ABB RAPID module: P401.mod

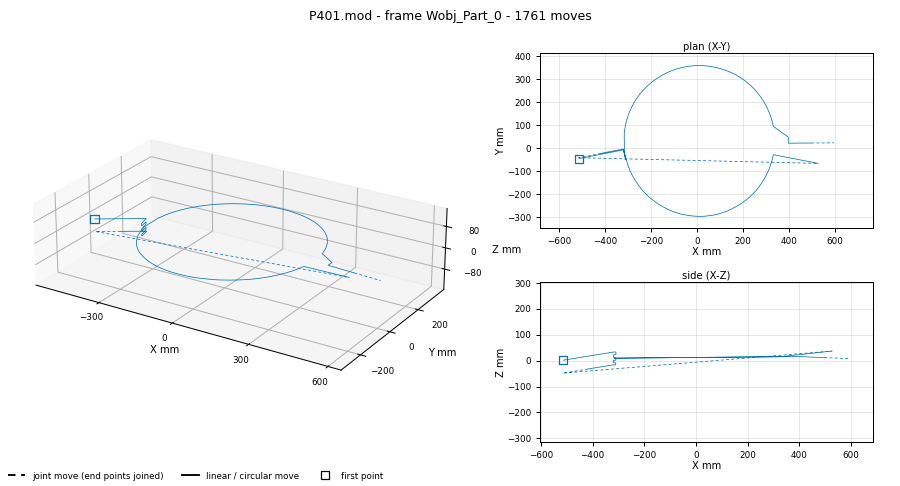
[picture p0: tool path of P401.mod in frame Wobj_Part_0, 1761 of 1771 moves have a stored position in this frame; points joined in program order, loops and branches not executed]
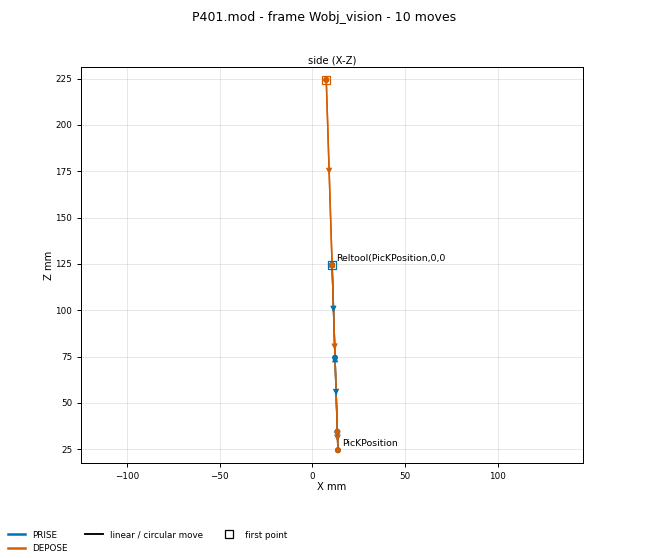
[picture p1: tool path of P401.mod in frame Wobj_vision, 10 of 1771 moves have a stored position in this frame; points joined in program order, loops and branches not executed]
MODULE P401

    ! Nom         :P401
    ! Description :
    ! Créé le     :07/06/2023 14:41:53

    LOCAL CONST SPEEDDATA VitesseLente :=[10,500,0,0];
	LOCAL CONST SPEEDDATA VitesseRapide :=[30,500,0,0];
	LOCAL CONST SPEEDDATA VitesseTronconnage :=[2,500,0,0];
	LOCAL CONST SPEEDDATA VitesseTronconnageApp :=[10,500,0,0];
    !
    !Point de prise
    LOCAL PERS Robtarget PicKPosition := [[13.7351915229446,28.8988205963881,24.4259709392431],[0.015425718644535,0.66713477772881,0.744749815337416,0.00639907055097392],[0,0,0,0],[8.999999E+09,8.999999E+09,8.999999E+09,8.999999E+09,8.999999E+09,8.999999E+09]];
	LOCAL PERS Pose Ref := [[0,0,0],[1,0,0,0]];
    !
    !Declaration des points de meulage

    !Tr_meulage_motif_1 : Meulage d'un motif
    LOCAL CONST Robtarget Tr_meulage_motif_1_0 := [[-319.4905625,-7.31827685546875,33.72298046875],[0.588012732058927,-0.500859688362471,0.411836559206125,-0.483498963816164],[0,0,0,0],[8.999999E+09,8.999999E+09,8.999999E+09,8.999999E+09,8.999999E+09,8.999999E+09]];
    LOCAL CONST Robtarget Tr_meulage_motif_1_1 := [[-319.26584375,-8.29269921875,33.72351171875],[0.588012732058927,-0.500859688362471,0.411836559206125,-0.483498963816164],[0,0,0,0],[8.999999E+09,8.999999E+09,8.999999E+09,8.999999E+09,8.999999E+09,8.999999E+09]];
    LOCAL CONST Robtarget Tr_meulage_motif_1_2 := [[-319.041125,-9.26712109375,33.72404296875],[0.588012732058927,-0.500859688362471,0.411836559206125,-0.483498963816164],[0,0,0,0],[8.999999E+09,8.999999E+09,8.999999E+09,8.999999E+09,8.999999E+09,8.999999E+09]];
    LOCAL CONST Robtarget Tr_meulage_motif_1_3 := [[-318.81640625,-10.24154296875,33.72457421875],[0.588012732058927,-0.500859688362471,0.411836559206125,-0.483498963816164],[0,0,0,0],[8.999999E+09,8.999999E+09,8.999999E+09,8.999999E+09,8.999999E+09,8.999999E+09]];
    LOCAL CONST Robtarget Tr_meulage_motif_1_4 := [[-318.59165625,-11.21596484375,33.725109375],[0.588012732058927,-0.500859688362471,0.411836559206125,-0.483498963816164],[0,0,0,0],[8.999999E+09,8.999999E+09,8.999999E+09,8.999999E+09,8.999999E+09,8.999999E+09]];
    LOCAL CONST Robtarget Tr_meulage_motif_1_5 := [[-318.3669375,-12.1903876953125,33.725640625],[0.588012732058927,-0.500859688362471,0.411836559206125,-0.483498963816164],[0,0,0,0],[8.999999E+09,8.999999E+09,8.999999E+09,8.999999E+09,8.999999E+09,8.999999E+09]];
    LOCAL CONST Robtarget Tr_meulage_motif_1_6 := [[-318.14221875,-13.1648095703125,33.726171875],[0.588012732058927,-0.500859688362471,0.411836559206125,-0.483498963816164],[0,0,0,0],[8.999999E+09,8.999999E+09,8.999999E+09,8.999999E+09,8.999999E+09,8.999999E+09]];
    LOCAL CONST Robtarget Tr_meulage_motif_1_7 := [[-317.9175,-14.1392314453125,33.726703125],[0.588012732058927,-0.500859688362471,0.411836559206125,-0.483498963816164],[0,0,0,0],[8.999999E+09,8.999999E+09,8.999999E+09,8.999999E+09,8.999999E+09,8.999999E+09]];
    LOCAL CONST Robtarget Tr_meulage_motif_1_8 := [[-317.69278125,-15.1136533203125,33.727234375],[0.588012732058927,-0.500859688362471,0.411836559206125,-0.483498963816164],[0,0,0,0],[8.999999E+09,8.999999E+09,8.999999E+09,8.999999E+09,8.999999E+09,8.999999E+09]];
    LOCAL CONST Robtarget Tr_meulage_motif_1_9 := [[-317.46803125,-16.0880751953125,33.72776953125],[0.588012732058927,-0.500859688362471,0.411836559206125,-0.483498963816164],[0,0,0,0],[8.999999E+09,8.999999E+09,8.999999E+09,8.999999E+09,8.999999E+09,8.999999E+09]];
    LOCAL CONST Robtarget Tr_meulage_motif_1_10 := [[-317.2433125,-17.062498046875,33.72830078125],[0.588012732058927,-0.500859688362471,0.411836559206125,-0.483498963816164],[0,0,0,0],[8.999999E+09,8.999999E+09,8.999999E+09,8.999999E+09,8.999999E+09,8.999999E+09]];
    LOCAL CONST Robtarget Tr_meulage_motif_1_11 := [[-317.01859375,-18.036919921875,33.72883203125],[0.588012732058927,-0.500859688362471,0.411836559206125,-0.483498963816164],[0,0,0,0],[8.999999E+09,8.999999E+09,8.999999E+09,8.999999E+09,8.999999E+09,8.999999E+09]];
    LOCAL CONST Robtarget Tr_meulage_motif_1_12 := [[-316.793875,-19.011341796875,33.72936328125],[0.588012732058927,-0.500859688362471,0.411836559206125,-0.483498963816164],[0,0,0,0],[8.999999E+09,8.999999E+09,8.999999E+09,8.999999E+09,8.999999E+09,8.999999E+09]];
    LOCAL CONST Robtarget Tr_meulage_motif_1_13 := [[-316.56915625,-19.985763671875,33.7298984375],[0.588012732058927,-0.500859688362471,0.411836559206125,-0.483498963816164],[0,0,0,0],[8.999999E+09,8.999999E+09,8.999999E+09,8.999999E+09,8.999999E+09,8.999999E+09]];
    LOCAL CONST Robtarget Tr_meulage_motif_1_14 := [[-316.34440625,-20.960185546875,33.7304296875],[0.588012732058927,-0.500859688362471,0.411836559206125,-0.483498963816164],[0,0,0,0],[8.999999E+09,8.999999E+09,8.999999E+09,8.999999E+09,8.999999E+09,8.999999E+09]];
    LOCAL CONST Robtarget Tr_meulage_motif_1_15 := [[-316.1196875,-21.934607421875,33.7309609375],[0.588012732058927,-0.500859688362471,0.411836559206125,-0.483498963816164],[0,0,0,0],[8.999999E+09,8.999999E+09,8.999999E+09,8.999999E+09,8.999999E+09,8.999999E+09]];
    LOCAL CONST Robtarget Tr_meulage_motif_1_16 := [[-315.89496875,-22.909029296875,33.7314921875],[0.588012732058927,-0.500859688362471,0.411836559206125,-0.483498963816164],[0,0,0,0],[8.999999E+09,8.999999E+09,8.999999E+09,8.999999E+09,8.999999E+09,8.999999E+09]];
    LOCAL CONST Robtarget Tr_meulage_motif_1_17 := [[-315.67025,-23.883451171875,33.73202734375],[0.588012732058927,-0.500859688362471,0.411836559206125,-0.483498963816164],[0,0,0,0],[8.999999E+09,8.999999E+09,8.999999E+09,8.999999E+09,8.999999E+09,8.999999E+09]];
    LOCAL CONST Robtarget Tr_meulage_motif_1_18 := [[-315.44553125,-24.857875,33.73255859375],[0.588012732058927,-0.500859688362471,0.411836559206125,-0.483498963816164],[0,0,0,0],[8.999999E+09,8.999999E+09,8.999999E+09,8.999999E+09,8.999999E+09,8.999999E+09]];
    LOCAL CONST Robtarget Tr_meulage_motif_1_19 := [[-315.22078125,-25.832296875,33.73308984375],[0.588012732058927,-0.500859688362471,0.411836559206125,-0.483498963816164],[0,0,0,0],[8.999999E+09,8.999999E+09,8.999999E+09,8.999999E+09,8.999999E+09,8.999999E+09]];
    LOCAL CONST Robtarget Tr_meulage_motif_1_20 := [[-314.9960625,-26.80671875,33.73362109375],[0.588012732058927,-0.500859688362471,0.411836559206125,-0.483498963816164],[0,0,0,0],[8.999999E+09,8.999999E+09,8.999999E+09,8.999999E+09,8.999999E+09,8.999999E+09]];
    LOCAL CONST Robtarget Tr_meulage_motif_1_21 := [[-314.77134375,-27.781140625,33.73415234375],[0.588012732058927,-0.500859688362471,0.411836559206125,-0.483498963816164],[0,0,0,0],[8.999999E+09,8.999999E+09,8.999999E+09,8.999999E+09,8.999999E+09,8.999999E+09]];
    LOCAL CONST Robtarget Tr_meulage_motif_1_22 := [[-314.546625,-28.7555625,33.7346875],[0.588012732058927,-0.500859688362471,0.411836559206125,-0.483498963816164],[0,0,0,0],[8.999999E+09,8.999999E+09,8.999999E+09,8.999999E+09,8.999999E+09,8.999999E+09]];
    LOCAL CONST Robtarget Tr_meulage_motif_1_23 := [[-314.32190625,-29.729984375,33.73521875],[0.588012732058927,-0.500859688362471,0.411836559206125,-0.483498963816164],[0,0,0,0],[8.999999E+09,8.999999E+09,8.999999E+09,8.999999E+09,8.999999E+09,8.999999E+09]];
    LOCAL CONST Robtarget Tr_meulage_motif_1_24 := [[-314.09715625,-30.70440625,33.73575],[0.588012732058927,-0.500859688362471,0.411836559206125,-0.483498963816164],[0,0,0,0],[8.999999E+09,8.999999E+09,8.999999E+09,8.999999E+09,8.999999E+09,8.999999E+09]];
    LOCAL CONST Robtarget Tr_meulage_motif_1_25 := [[-313.8724375,-31.678828125,33.73628125],[0.588012732058927,-0.500859688362471,0.411836559206125,-0.483498963816164],[0,0,0,0],[8.999999E+09,8.999999E+09,8.999999E+09,8.999999E+09,8.999999E+09,8.999999E+09]];
    LOCAL CONST Robtarget Tr_meulage_motif_1_26 := [[-313.64771875,-32.65325,33.73681640625],[0.588012732058927,-0.500859688362471,0.411836559206125,-0.483498963816164],[0,0,0,0],[8.999999E+09,8.999999E+09,8.999999E+09,8.999999E+09,8.999999E+09,8.999999E+09]];
    LOCAL CONST Robtarget Tr_meulage_motif_1_27 := [[-313.423,-33.627671875,33.73734765625],[0.588012732058927,-0.500859688362471,0.411836559206125,-0.483498963816164],[0,0,0,0],[8.999999E+09,8.999999E+09,8.999999E+09,8.999999E+09,8.999999E+09,8.999999E+09]];
    LOCAL CONST Robtarget Tr_meulage_motif_1_28 := [[-313.19828125,-34.60209375,33.73787890625],[0.588012732058927,-0.500859688362471,0.411836559206125,-0.483498963816164],[0,0,0,0],[8.999999E+09,8.999999E+09,8.999999E+09,8.999999E+09,8.999999E+09,8.999999E+09]];
    LOCAL CONST Robtarget Tr_meulage_motif_1_29 := [[-312.97353125,-35.576515625,33.73841015625],[0.588012732058927,-0.500859688362471,0.411836559206125,-0.483498963816164],[0,0,0,0],[8.999999E+09,8.999999E+09,8.999999E+09,8.999999E+09,8.999999E+09,8.999999E+09]];
    LOCAL CONST Robtarget Tr_meulage_motif_1_30 := [[-312.7488125,-36.5509375,33.73894140625],[0.588012732058927,-0.500859688362471,0.411836559206125,-0.483498963816164],[0,0,0,0],[8.999999E+09,8.999999E+09,8.999999E+09,8.999999E+09,8.999999E+09,8.999999E+09]];
    LOCAL CONST Robtarget Tr_meulage_motif_1_31 := [[-312.52409375,-37.525359375,33.7394765625],[0.588012732058927,-0.500859688362471,0.411836559206125,-0.483498963816164],[0,0,0,0],[8.999999E+09,8.999999E+09,8.999999E+09,8.999999E+09,8.999999E+09,8.999999E+09]];
    LOCAL CONST Robtarget Tr_meulage_motif_1_32 := [[-312.299375,-38.49978125,33.7400078125],[0.588012732058927,-0.500859688362471,0.411836559206125,-0.483498963816164],[0,0,0,0],[8.999999E+09,8.999999E+09,8.999999E+09,8.999999E+09,8.999999E+09,8.999999E+09]];
    LOCAL CONST Robtarget Tr_meulage_motif_1_33 := [[-312.07465625,-39.47420703125,33.7405390625],[0.588012732058927,-0.500859688362471,0.411836559206125,-0.483498963816164],[0,0,0,0],[8.999999E+09,8.999999E+09,8.999999E+09,8.999999E+09,8.999999E+09,8.999999E+09]];
    LOCAL CONST Robtarget Tr_meulage_motif_1_34 := [[-311.84990625,-40.44862890625,33.7410703125],[0.588012732058927,-0.500859688362471,0.411836559206125,-0.483498963816164],[0,0,0,0],[8.999999E+09,8.999999E+09,8.999999E+09,8.999999E+09,8.999999E+09,8.999999E+09]];
    LOCAL CONST Robtarget Tr_meulage_motif_1_35 := [[-311.6251875,-41.42305078125,33.74160546875],[0.588012732058927,-0.500859688362471,0.411836559206125,-0.483498963816164],[0,0,0,0],[8.999999E+09,8.999999E+09,8.999999E+09,8.999999E+09,8.999999E+09,8.999999E+09]];
    LOCAL CONST Robtarget Tr_meulage_motif_1_36 := [[-311.40046875,-42.39747265625,33.74213671875],[0.588012732058927,-0.500859688362471,0.411836559206125,-0.483498963816164],[0,0,0,0],[8.999999E+09,8.999999E+09,8.999999E+09,8.999999E+09,8.999999E+09,8.999999E+09]];
    LOCAL CONST Robtarget Tr_meulage_motif_1_37 := [[-311.17575,-43.37189453125,33.74266796875],[0.588012732058927,-0.500859688362471,0.411836559206125,-0.483498963816164],[0,0,0,0],[8.999999E+09,8.999999E+09,8.999999E+09,8.999999E+09,8.999999E+09,8.999999E+09]];
    LOCAL CONST Robtarget Tr_meulage_motif_1_38 := [[-310.95103125,-44.34631640625,33.74319921875],[0.588012732058927,-0.500859688362471,0.411836559206125,-0.483498963816164],[0,0,0,0],[8.999999E+09,8.999999E+09,8.999999E+09,8.999999E+09,8.999999E+09,8.999999E+09]];
    LOCAL CONST Robtarget Tr_meulage_motif_1_39 := [[-310.72928125,-45.31385546875,33.63314453125],[0.588012732058927,-0.500859688362471,0.411836559206125,-0.483498963816164],[0,0,0,0],[8.999999E+09,8.999999E+09,8.999999E+09,8.999999E+09,8.999999E+09,8.999999E+09]];
    LOCAL CONST Robtarget Tr_meulage_motif_1_40 := [[-310.51909375,-46.23683984375,33.4224765625],[0.588012732058927,-0.500859688362471,0.411836559206125,-0.483498963816164],[0,0,0,0],[8.999999E+09,8.999999E+09,8.999999E+09,8.999999E+09,8.999999E+09,8.999999E+09]];
    LOCAL CONST Robtarget Tr_meulage_motif_1_41 := [[-310.3306875,-47.06864453125,33.15110546875],[0.588012732058927,-0.500859688362471,0.411836559206125,-0.483498963816164],[0,0,0,0],[8.999999E+09,8.999999E+09,8.999999E+09,8.999999E+09,8.999999E+09,8.999999E+09]];
    LOCAL CONST Robtarget Tr_meulage_motif_1_42 := [[-310.16546875,-47.8003046875,32.87558984375],[0.588012732058927,-0.500859688362471,0.411836559206125,-0.483498963816164],[0,0,0,0],[8.999999E+09,8.999999E+09,8.999999E+09,8.999999E+09,8.999999E+09,8.999999E+09]];
    LOCAL CONST Robtarget Tr_meulage_motif_1_43 := [[-309.92534375,-48.875234375,32.26009765625],[0.588012732058927,-0.500859688362471,0.411836559206125,-0.483498963816164],[0,0,0,0],[8.999999E+09,8.999999E+09,8.999999E+09,8.999999E+09,8.999999E+09,8.999999E+09]];
    LOCAL CONST Robtarget Tr_meulage_motif_1_44 := [[-309.70534375,-49.8757109375,31.41305078125],[0.588012732058927,-0.500859688362471,0.411836559206125,-0.483498963816164],[0,0,0,0],[8.999999E+09,8.999999E+09,8.999999E+09,8.999999E+09,8.999999E+09,8.999999E+09]];
    LOCAL CONST Robtarget Tr_meulage_motif_1_45 := [[-309.5270625,-50.7050546875,30.389705078125],[0.588012732058927,-0.500859688362471,0.411836559206125,-0.483498963816164],[0,0,0,0],[8.999999E+09,8.999999E+09,8.999999E+09,8.999999E+09,8.999999E+09,8.999999E+09]];
    LOCAL CONST Robtarget Tr_meulage_motif_1_46 := [[-309.430625,-51.1843984375,29.273861328125],[0.588012732058927,-0.500859688362471,0.411836559206125,-0.483498963816164],[0,0,0,0],[8.999999E+09,8.999999E+09,8.999999E+09,8.999999E+09,8.999999E+09,8.999999E+09]];
    LOCAL CONST Robtarget Tr_meulage_motif_1_47 := [[-309.43284375,-51.2130625,28.5779609375],[0.588012732058927,-0.500859688362471,0.411836559206125,-0.483498963816164],[0,0,0,0],[8.999999E+09,8.999999E+09,8.999999E+09,8.999999E+09,8.999999E+09,8.999999E+09]];
    LOCAL CONST Robtarget Tr_meulage_motif_1_48 := [[-309.44071875,-51.21523828125,27.91676171875],[0.588012732058927,-0.500859688362471,0.411836559206125,-0.483498963816164],[0,0,0,0],[8.999999E+09,8.999999E+09,8.999999E+09,8.999999E+09,8.999999E+09,8.999999E+09]];
    LOCAL CONST Robtarget Tr_meulage_motif_1_49 := [[-309.46090625,-51.16394140625,27.2556875],[0.588012732058927,-0.500859688362471,0.411836559206125,-0.483498963816164],[0,0,0,0],[8.999999E+09,8.999999E+09,8.999999E+09,8.999999E+09,8.999999E+09,8.999999E+09]];
    LOCAL CONST Robtarget Tr_meulage_motif_1_50 := [[-309.586,-50.68209375,26.1537578125],[0.588012732058927,-0.500859688362471,0.411836559206125,-0.483498963816164],[0,0,0,0],[8.999999E+09,8.999999E+09,8.999999E+09,8.999999E+09,8.999999E+09,8.999999E+09]];
    LOCAL CONST Robtarget Tr_meulage_motif_1_51 := [[-309.79046875,-49.85069140625,25.14675390625],[0.588012732058927,-0.500859688362471,0.411836559206125,-0.483498963816164],[0,0,0,0],[8.999999E+09,8.999999E+09,8.999999E+09,8.999999E+09,8.999999E+09,8.999999E+09]];
    LOCAL CONST Robtarget Tr_meulage_motif_1_52 := [[-310.03034375,-48.85619140625,24.317396484375],[0.588012732058927,-0.500859688362471,0.411836559206125,-0.483498963816164],[0,0,0,0],[8.999999E+09,8.999999E+09,8.999999E+09,8.999999E+09,8.999999E+09,8.999999E+09]];
    LOCAL CONST Robtarget Tr_meulage_motif_1_53 := [[-310.1894375,-48.18797265625,23.921310546875],[0.588012732058927,-0.500859688362471,0.411836559206125,-0.483498963816164],[0,0,0,0],[8.999999E+09,8.999999E+09,8.999999E+09,8.999999E+09,8.999999E+09,8.999999E+09]];
    LOCAL CONST Robtarget Tr_meulage_motif_1_54 := [[-310.45553125,-47.061046875,23.433201171875],[0.588012732058927,-0.500859688362471,0.411836559206125,-0.483498963816164],[0,0,0,0],[8.999999E+09,8.999999E+09,8.999999E+09,8.999999E+09,8.999999E+09,8.999999E+09]];
    LOCAL CONST Robtarget Tr_meulage_motif_1_55 := [[-310.6485625,-46.23849609375,23.168677734375],[0.588012732058927,-0.500859688362471,0.411836559206125,-0.483498963816164],[0,0,0,0],[8.999999E+09,8.999999E+09,8.999999E+09,8.999999E+09,8.999999E+09,8.999999E+09]];
    LOCAL CONST Robtarget Tr_meulage_motif_1_56 := [[-310.8604375,-45.3310078125,22.963728515625],[0.588012732058927,-0.500859688362471,0.411836559206125,-0.483498963816164],[0,0,0,0],[8.999999E+09,8.999999E+09,8.999999E+09,8.999999E+09,8.999999E+09,8.999999E+09]];
    LOCAL CONST Robtarget Tr_meulage_motif_1_57 := [[-311.0823125,-44.37491015625,22.85462109375],[0.588012732058927,-0.500859688362471,0.411836559206125,-0.483498963816164],[0,0,0,0],[8.999999E+09,8.999999E+09,8.999999E+09,8.999999E+09,8.999999E+09,8.999999E+09]];
    LOCAL CONST Robtarget Tr_meulage_motif_1_58 := [[-311.3066875,-43.4081015625,22.7435078125],[0.588012732058927,-0.500859688362471,0.411836559206125,-0.483498963816164],[0,0,0,0],[8.999999E+09,8.999999E+09,8.999999E+09,8.999999E+09,8.999999E+09,8.999999E+09]];
    LOCAL CONST Robtarget Tr_meulage_motif_1_59 := [[-311.53140625,-42.4336796875,22.742974609375],[0.588012732058927,-0.500859688362471,0.411836559206125,-0.483498963816164],[0,0,0,0],[8.999999E+09,8.999999E+09,8.999999E+09,8.999999E+09,8.999999E+09,8.999999E+09]];
    LOCAL CONST Robtarget Tr_meulage_motif_1_60 := [[-311.756125,-41.4592578125,22.742443359375],[0.588012732058927,-0.500859688362471,0.411836559206125,-0.483498963816164],[0,0,0,0],[8.999999E+09,8.999999E+09,8.999999E+09,8.999999E+09,8.999999E+09,8.999999E+09]];
    LOCAL CONST Robtarget Tr_meulage_motif_1_61 := [[-311.980875,-40.48483203125,22.74191015625],[0.588012732058927,-0.500859688362471,0.411836559206125,-0.483498963816164],[0,0,0,0],[8.999999E+09,8.999999E+09,8.999999E+09,8.999999E+09,8.999999E+09,8.999999E+09]];
    LOCAL CONST Robtarget Tr_meulage_motif_1_62 := [[-312.20559375,-39.51041015625,22.74137890625],[0.588012732058927,-0.500859688362471,0.411836559206125,-0.483498963816164],[0,0,0,0],[8.999999E+09,8.999999E+09,8.999999E+09,8.999999E+09,8.999999E+09,8.999999E+09]];
    LOCAL CONST Robtarget Tr_meulage_motif_1_63 := [[-312.4303125,-38.53598828125,22.740845703125],[0.588012732058927,-0.500859688362471,0.411836559206125,-0.483498963816164],[0,0,0,0],[8.999999E+09,8.999999E+09,8.999999E+09,8.999999E+09,8.999999E+09,8.999999E+09]];
    LOCAL CONST Robtarget Tr_meulage_motif_1_64 := [[-312.65503125,-37.56156640625,22.740314453125],[0.588012732058927,-0.500859688362471,0.411836559206125,-0.483498963816164],[0,0,0,0],[8.999999E+09,8.999999E+09,8.999999E+09,8.999999E+09,8.999999E+09,8.999999E+09]];
    LOCAL CONST Robtarget Tr_meulage_motif_1_65 := [[-312.87975,-36.58714453125,22.739783203125],[0.588012732058927,-0.500859688362471,0.411836559206125,-0.483498963816164],[0,0,0,0],[8.999999E+09,8.999999E+09,8.999999E+09,8.999999E+09,8.999999E+09,8.999999E+09]];
    LOCAL CONST Robtarget Tr_meulage_motif_1_66 := [[-313.1045,-35.61272265625,22.73925],[0.588012732058927,-0.500859688362471,0.411836559206125,-0.483498963816164],[0,0,0,0],[8.999999E+09,8.999999E+09,8.999999E+09,8.999999E+09,8.999999E+09,8.999999E+09]];
    LOCAL CONST Robtarget Tr_meulage_motif_1_67 := [[-313.32921875,-34.63830078125,22.73871875],[0.588012732058927,-0.500859688362471,0.411836559206125,-0.483498963816164],[0,0,0,0],[8.999999E+09,8.999999E+09,8.999999E+09,8.999999E+09,8.999999E+09,8.999999E+09]];
    LOCAL CONST Robtarget Tr_meulage_motif_1_68 := [[-313.5539375,-33.66387890625,22.738185546875],[0.588012732058927,-0.500859688362471,0.411836559206125,-0.483498963816164],[0,0,0,0],[8.999999E+09,8.999999E+09,8.999999E+09,8.999999E+09,8.999999E+09,8.999999E+09]];
    LOCAL CONST Robtarget Tr_meulage_motif_1_69 := [[-313.77865625,-32.68945703125,22.737654296875],[0.588012732058927,-0.500859688362471,0.411836559206125,-0.483498963816164],[0,0,0,0],[8.999999E+09,8.999999E+09,8.999999E+09,8.999999E+09,8.999999E+09,8.999999E+09]];
    LOCAL CONST Robtarget Tr_meulage_motif_1_70 := [[-314.003375,-31.71503515625,22.73712109375],[0.588012732058927,-0.500859688362471,0.411836559206125,-0.483498963816164],[0,0,0,0],[8.999999E+09,8.999999E+09,8.999999E+09,8.999999E+09,8.999999E+09,8.999999E+09]];
    LOCAL CONST Robtarget Tr_meulage_motif_1_71 := [[-314.228125,-30.74061328125,22.73658984375],[0.588012732058927,-0.500859688362471,0.411836559206125,-0.483498963816164],[0,0,0,0],[8.999999E+09,8.999999E+09,8.999999E+09,8.999999E+09,8.999999E+09,8.999999E+09]];
    LOCAL CONST Robtarget Tr_meulage_motif_1_72 := [[-314.45284375,-29.76619140625,22.736056640625],[0.588012732058927,-0.500859688362471,0.411836559206125,-0.483498963816164],[0,0,0,0],[8.999999E+09,8.999999E+09,8.999999E+09,8.999999E+09,8.999999E+09,8.999999E+09]];
    LOCAL CONST Robtarget Tr_meulage_motif_1_73 := [[-314.6775625,-28.79176953125,22.735525390625],[0.588012732058927,-0.500859688362471,0.411836559206125,-0.483498963816164],[0,0,0,0],[8.999999E+09,8.999999E+09,8.999999E+09,8.999999E+09,8.999999E+09,8.999999E+09]];
    LOCAL CONST Robtarget Tr_meulage_motif_1_74 := [[-314.90228125,-27.81734765625,22.7349921875],[0.588012732058927,-0.500859688362471,0.411836559206125,-0.483498963816164],[0,0,0,0],[8.999999E+09,8.999999E+09,8.999999E+09,8.999999E+09,8.999999E+09,8.999999E+09]];
    LOCAL CONST Robtarget Tr_meulage_motif_1_75 := [[-315.12703125,-26.84292578125,22.7344609375],[0.588012732058927,-0.500859688362471,0.411836559206125,-0.483498963816164],[0,0,0,0],[8.999999E+09,8.999999E+09,8.999999E+09,8.999999E+09,8.999999E+09,8.999999E+09]];
    LOCAL CONST Robtarget Tr_meulage_motif_1_76 := [[-315.35175,-25.868501953125,22.7339296875],[0.588012732058927,-0.500859688362471,0.411836559206125,-0.483498963816164],[0,0,0,0],[8.999999E+09,8.999999E+09,8.999999E+09,8.999999E+09,8.999999E+09,8.999999E+09]];
    LOCAL CONST Robtarget Tr_meulage_motif_1_77 := [[-315.57646875,-24.894080078125,22.733396484375],[0.588012732058927,-0.500859688362471,0.411836559206125,-0.483498963816164],[0,0,0,0],[8.999999E+09,8.999999E+09,8.999999E+09,8.999999E+09,8.999999E+09,8.999999E+09]];
    LOCAL CONST Robtarget Tr_meulage_motif_1_78 := [[-315.8011875,-23.919658203125,22.732865234375],[0.588012732058927,-0.500859688362471,0.411836559206125,-0.483498963816164],[0,0,0,0],[8.999999E+09,8.999999E+09,8.999999E+09,8.999999E+09,8.999999E+09,8.999999E+09]];
    LOCAL CONST Robtarget Tr_meulage_motif_1_79 := [[-316.02590625,-22.945236328125,22.73233203125],[0.588012732058927,-0.500859688362471,0.411836559206125,-0.483498963816164],[0,0,0,0],[8.999999E+09,8.999999E+09,8.999999E+09,8.999999E+09,8.999999E+09,8.999999E+09]];
    LOCAL CONST Robtarget Tr_meulage_motif_1_80 := [[-316.25065625,-21.970814453125,22.73180078125],[0.588012732058927,-0.500859688362471,0.411836559206125,-0.483498963816164],[0,0,0,0],[8.999999E+09,8.999999E+09,8.999999E+09,8.999999E+09,8.999999E+09,8.999999E+09]];
    LOCAL CONST Robtarget Tr_meulage_motif_1_81 := [[-316.475375,-20.996392578125,22.731267578125],[0.588012732058927,-0.500859688362471,0.411836559206125,-0.483498963816164],[0,0,0,0],[8.999999E+09,8.999999E+09,8.999999E+09,8.999999E+09,8.999999E+09,8.999999E+09]];
    LOCAL CONST Robtarget Tr_meulage_motif_1_82 := [[-316.70009375,-20.021970703125,22.730736328125],[0.588012732058927,-0.500859688362471,0.411836559206125,-0.483498963816164],[0,0,0,0],[8.999999E+09,8.999999E+09,8.999999E+09,8.999999E+09,8.999999E+09,8.999999E+09]];
    LOCAL CONST Robtarget Tr_meulage_motif_1_83 := [[-316.9248125,-19.047548828125,22.730203125],[0.588012732058927,-0.500859688362471,0.411836559206125,-0.483498963816164],[0,0,0,0],[8.999999E+09,8.999999E+09,8.999999E+09,8.999999E+09,8.999999E+09,8.999999E+09]];
    LOCAL CONST Robtarget Tr_meulage_motif_1_84 := [[-317.14953125,-18.073126953125,22.729671875],[0.588012732058927,-0.500859688362471,0.411836559206125,-0.483498963816164],[0,0,0,0],[8.999999E+09,8.999999E+09,8.999999E+09,8.999999E+09,8.999999E+09,8.999999E+09]];
    LOCAL CONST Robtarget Tr_meulage_motif_1_85 := [[-317.37428125,-17.098705078125,22.729138671875],[0.588012732058927,-0.500859688362471,0.411836559206125,-0.483498963816164],[0,0,0,0],[8.999999E+09,8.999999E+09,8.999999E+09,8.999999E+09,8.999999E+09,8.999999E+09]];
    LOCAL CONST Robtarget Tr_meulage_motif_1_86 := [[-317.599,-16.1242822265625,22.728607421875],[0.588012732058927,-0.500859688362471,0.411836559206125,-0.483498963816164],[0,0,0,0],[8.999999E+09,8.999999E+09,8.999999E+09,8.999999E+09,8.999999E+09,8.999999E+09]];
    LOCAL CONST Robtarget Tr_meulage_motif_1_87 := [[-317.82371875,-15.1498603515625,22.72807421875],[0.588012732058927,-0.500859688362471,0.411836559206125,-0.483498963816164],[0,0,0,0],[8.999999E+09,8.999999E+09,8.999999E+09,8.999999E+09,8.999999E+09,8.999999E+09]];
    LOCAL CONST Robtarget Tr_meulage_motif_1_88 := [[-318.0484375,-14.1754384765625,22.72754296875],[0.588012732058927,-0.500859688362471,0.411836559206125,-0.483498963816164],[0,0,0,0],[8.999999E+09,8.999999E+09,8.999999E+09,8.999999E+09,8.999999E+09,8.999999E+09]];
    LOCAL CONST Robtarget Tr_meulage_motif_1_89 := [[-318.2728125,-13.208626953125,22.6164296875],[0.588012732058927,-0.500859688362471,0.411836559206125,-0.483498963816164],[0,0,0,0],[8.999999E+09,8.999999E+09,8.999999E+09,8.999999E+09,8.999999E+09,8.999999E+09]];
    LOCAL CONST Robtarget Tr_meulage_motif_1_90 := [[-318.48803125,-12.2870322265625,22.40475390625],[0.588012732058927,-0.500859688362471,0.411836559206125,-0.483498963816164],[0,0,0,0],[8.999999E+09,8.999999E+09,8.999999E+09,8.999999E+09,8.999999E+09,8.999999E+09]];
    LOCAL CONST Robtarget Tr_meulage_motif_1_91 := [[-318.68290625,-11.4570185546875,22.132478515625],[0.588012732058927,-0.500859688362471,0.411836559206125,-0.483498963816164],[0,0,0,0],[8.999999E+09,8.999999E+09,8.999999E+09,8.999999E+09,8.999999E+09,8.999999E+09]];
    LOCAL CONST Robtarget Tr_meulage_motif_1_92 := [[-318.84640625,-10.76471875,21.827966796875],[0.588012732058927,-0.500859688362471,0.411836559206125,-0.483498963816164],[0,0,0,0],[8.999999E+09,8.999999E+09,8.999999E+09,8.999999E+09,8.999999E+09,8.999999E+09]];
    LOCAL CONST Robtarget Tr_meulage_motif_1_93 := [[-319.08675,-9.758890625,21.164935546875],[0.588012732058927,-0.500859688362471,0.411836559206125,-0.483498963816164],[0,0,0,0],[8.999999E+09,8.999999E+09,8.999999E+09,8.999999E+09,8.999999E+09,8.999999E+09]];
    LOCAL CONST Robtarget Tr_meulage_motif_1_94 := [[-319.3001875,-8.8829912109375,20.2625859375],[0.588012732058927,-0.500859688362471,0.411836559206125,-0.483498963816164],[0,0,0,0],[8.999999E+09,8.999999E+09,8.999999E+09,8.999999E+09,8.999999E+09,8.999999E+09]];
    LOCAL CONST Robtarget Tr_meulage_motif_1_95 := [[-319.432875,-8.3651484375,19.216349609375],[0.588012732058927,-0.500859688362471,0.411836559206125,-0.483498963816164],[0,0,0,0],[8.999999E+09,8.999999E+09,8.999999E+09,8.999999E+09,8.999999E+09,8.999999E+09]];
    LOCAL CONST Robtarget Tr_meulage_motif_1_96 := [[-319.482625,-8.18737548828125,18.5230859375],[0.588012732058927,-0.500859688362471,0.411836559206125,-0.483498963816164],[0,0,0,0],[8.999999E+09,8.999999E+09,8.999999E+09,8.999999E+09,8.999999E+09,8.999999E+09]];
    LOCAL CONST Robtarget Tr_meulage_motif_1_97 := [[-319.50615625,-8.12769921875,17.753111328125],[0.588012732058927,-0.500859688362471,0.411836559206125,-0.483498963816164],[0,0,0,0],[8.999999E+09,8.999999E+09,8.999999E+09,8.999999E+09,8.999999E+09,8.999999E+09]];
    LOCAL CONST Robtarget Tr_meulage_motif_1_98 := [[-319.50028125,-8.195458984375,16.983330078125],[0.588012732058927,-0.500859688362471,0.411836559206125,-0.483498963816164],[0,0,0,0],[8.999999E+09,8.999999E+09,8.999999E+09,8.999999E+09,8.999999E+09,8.999999E+09]];
    LOCAL CONST Robtarget Tr_meulage_motif_1_99 := [[-319.4191875,-8.6079677734375,15.8753876953125],[0.588012732058927,-0.500859688362471,0.411836559206125,-0.483498963816164],[0,0,0,0],[8.999999E+09,8.999999E+09,8.999999E+09,8.999999E+09,8.999999E+09,8.999999E+09]];
    LOCAL CONST Robtarget Tr_meulage_motif_1_100 := [[-319.33303125,-9.013611328125,15.2899658203125],[0.588012732058927,-0.500859688362471,0.411836559206125,-0.483498963816164],[0,0,0,0],[8.999999E+09,8.999999E+09,8.999999E+09,8.999999E+09,8.999999E+09,8.999999E+09]];
    LOCAL CONST Robtarget Tr_meulage_motif_1_101 := [[-319.14425,-9.88096484375,14.4033798828125],[0.588012732058927,-0.500859688362471,0.411836559206125,-0.483498963816164],[0,0,0,0],[8.999999E+09,8.999999E+09,8.999999E+09,8.999999E+09,8.999999E+09,8.999999E+09]];
    LOCAL CONST Robtarget Tr_meulage_motif_1_102 := [[-319.0175625,-10.4530361328125,13.9894111328125],[0.588012732058927,-0.500859688362471,0.411836559206125,-0.483498963816164],[0,0,0,0],[8.999999E+09,8.999999E+09,8.999999E+09,8.999999E+09,8.999999E+09,8.999999E+09]];
    LOCAL CONST Robtarget Tr_meulage_motif_1_103 := [[-318.7728125,-11.544138671875,13.445953125],[0.588012732058927,-0.500859688362471,0.411836559206125,-0.483498963816164],[0,0,0,0],[8.999999E+09,8.999999E+09,8.999999E+09,8.999999E+09,8.999999E+09,8.999999E+09]];
    LOCAL CONST Robtarget Tr_meulage_motif_1_104 := [[-318.59078125,-12.3495888671875,13.1509150390625],[0.588012732058927,-0.500859688362471,0.411836559206125,-0.483498963816164],[0,0,0,0],[8.999999E+09,8.999999E+09,8.999999E+09,8.999999E+09,8.999999E+09,8.999999E+09]];
    LOCAL CONST Robtarget Tr_meulage_motif_1_105 := [[-318.38378125,-13.2584228515625,12.9469580078125],[0.588012732058927,-0.500859688362471,0.411836559206125,-0.483498963816164],[0,0,0,0],[8.999999E+09,8.999999E+09,8.999999E+09,8.999999E+09,8.999999E+09,8.999999E+09]];
    LOCAL CONST Robtarget Tr_meulage_motif_1_106 := [[-318.1645,-14.215236328125,12.8388955078125],[0.588012732058927,-0.500859688362471,0.411836559206125,-0.483498963816164],[0,0,0,0],[8.999999E+09,8.999999E+09,8.999999E+09,8.999999E+09,8.999999E+09,8.999999E+09]];
    LOCAL CONST Robtarget Tr_meulage_motif_1_107 := [[-317.94275,-15.182775390625,12.728837890625],[0.588012732058927,-0.500859688362471,0.411836559206125,-0.483498963816164],[0,0,0,0],[8.999999E+09,8.999999E+09,8.999999E+09,8.999999E+09,8.999999E+09,8.999999E+09]];
    LOCAL CONST Robtarget Tr_meulage_motif_1_108 := [[-317.71803125,-16.157197265625,12.7293701171875],[0.588012732058927,-0.500859688362471,0.411836559206125,-0.483498963816164],[0,0,0,0],[8.999999E+09,8.999999E+09,8.999999E+09,8.999999E+09,8.999999E+09,8.999999E+09]];
    LOCAL CONST Robtarget Tr_meulage_motif_1_109 := [[-317.4933125,-17.131619140625,12.72990234375],[0.588012732058927,-0.500859688362471,0.411836559206125,-0.483498963816164],[0,0,0,0],[8.999999E+09,8.999999E+09,8.999999E+09,8.999999E+09,8.999999E+09,8.999999E+09]];
    LOCAL CONST Robtarget Tr_meulage_motif_1_110 := [[-317.26859375,-18.106041015625,12.7304345703125],[0.588012732058927,-0.500859688362471,0.411836559206125,-0.483498963816164],[0,0,0,0],[8.999999E+09,8.999999E+09,8.999999E+09,8.999999E+09,8.999999E+09,8.999999E+09]];
    LOCAL CONST Robtarget Tr_meulage_motif_1_111 := [[-317.043875,-19.080462890625,12.730966796875],[0.588012732058927,-0.500859688362471,0.411836559206125,-0.483498963816164],[0,0,0,0],[8.999999E+09,8.999999E+09,8.999999E+09,8.999999E+09,8.999999E+09,8.999999E+09]];
    LOCAL CONST Robtarget Tr_meulage_motif_1_112 := [[-316.819125,-20.054884765625,12.7314990234375],[0.588012732058927,-0.500859688362471,0.411836559206125,-0.483498963816164],[0,0,0,0],[8.999999E+09,8.999999E+09,8.999999E+09,8.999999E+09,8.999999E+09,8.999999E+09]];
    LOCAL CONST Robtarget Tr_meulage_motif_1_113 := [[-316.59440625,-21.02930859375,12.73203125],[0.588012732058927,-0.500859688362471,0.411836559206125,-0.483498963816164],[0,0,0,0],[8.999999E+09,8.999999E+09,8.999999E+09,8.999999E+09,8.999999E+09,8.999999E+09]];
    LOCAL CONST Robtarget Tr_meulage_motif_1_114 := [[-316.3696875,-22.00373046875,12.7325625],[0.588012732058927,-0.500859688362471,0.411836559206125,-0.483498963816164],[0,0,0,0],[8.999999E+09,8.999999E+09,8.999999E+09,8.999999E+09,8.999999E+09,8.999999E+09]];
    LOCAL CONST Robtarget Tr_meulage_motif_1_115 := [[-316.14496875,-22.97815234375,12.7330947265625],[0.588012732058927,-0.500859688362471,0.411836559206125,-0.483498963816164],[0,0,0,0],[8.999999E+09,8.999999E+09,8.999999E+09,8.999999E+09,8.999999E+09,8.999999E+09]];
    LOCAL CONST Robtarget Tr_meulage_motif_1_116 := [[-315.92025,-23.95257421875,12.733626953125],[0.588012732058927,-0.500859688362471,0.411836559206125,-0.483498963816164],[0,0,0,0],[8.999999E+09,8.999999E+09,8.999999E+09,8.999999E+09,8.999999E+09,8.999999E+09]];
    LOCAL CONST Robtarget Tr_meulage_motif_1_117 := [[-315.6955,-24.92699609375,12.7341591796875],[0.588012732058927,-0.500859688362471,0.411836559206125,-0.483498963816164],[0,0,0,0],[8.999999E+09,8.999999E+09,8.999999E+09,8.999999E+09,8.999999E+09,8.999999E+09]];
    LOCAL CONST Robtarget Tr_meulage_motif_1_118 := [[-315.47078125,-25.90141796875,12.73469140625],[0.588012732058927,-0.500859688362471,0.411836559206125,-0.483498963816164],[0,0,0,0],[8.999999E+09,8.999999E+09,8.999999E+09,8.999999E+09,8.999999E+09,8.999999E+09]];
    LOCAL CONST Robtarget Tr_meulage_motif_1_119 := [[-315.2460625,-26.87583984375,12.7352236328125],[0.588012732058927,-0.500859688362471,0.411836559206125,-0.483498963816164],[0,0,0,0],[8.999999E+09,8.999999E+09,8.999999E+09,8.999999E+09,8.999999E+09,8.999999E+09]];
    LOCAL CONST Robtarget Tr_meulage_motif_1_120 := [[-315.02134375,-27.85026171875,12.735755859375],[0.588012732058927,-0.500859688362471,0.411836559206125,-0.483498963816164],[0,0,0,0],[8.999999E+09,8.999999E+09,8.999999E+09,8.999999E+09,8.999999E+09,8.999999E+09]];
    LOCAL CONST Robtarget Tr_meulage_motif_1_121 := [[-314.796625,-28.82468359375,12.7362880859375],[0.588012732058927,-0.500859688362471,0.411836559206125,-0.483498963816164],[0,0,0,0],[8.999999E+09,8.999999E+09,8.999999E+09,8.999999E+09,8.999999E+09,8.999999E+09]];
    LOCAL CONST Robtarget Tr_meulage_motif_1_122 := [[-314.571875,-29.79910546875,12.7368203125],[0.588012732058927,-0.500859688362471,0.411836559206125,-0.483498963816164],[0,0,0,0],[8.999999E+09,8.999999E+09,8.999999E+09,8.999999E+09,8.999999E+09,8.999999E+09]];
    LOCAL CONST Robtarget Tr_meulage_motif_1_123 := [[-314.34715625,-30.77352734375,12.7373525390625],[0.588012732058927,-0.500859688362471,0.411836559206125,-0.483498963816164],[0,0,0,0],[8.999999E+09,8.999999E+09,8.999999E+09,8.999999E+09,8.999999E+09,8.999999E+09]];
    LOCAL CONST Robtarget Tr_meulage_motif_1_124 := [[-314.1224375,-31.747951171875,12.737884765625],[0.588012732058927,-0.500859688362471,0.411836559206125,-0.483498963816164],[0,0,0,0],[8.999999E+09,8.999999E+09,8.999999E+09,8.999999E+09,8.999999E+09,8.999999E+09]];
    LOCAL CONST Robtarget Tr_meulage_motif_1_125 := [[-313.89771875,-32.722373046875,12.7384169921875],[0.588012732058927,-0.500859688362471,0.411836559206125,-0.483498963816164],[0,0,0,0],[8.999999E+09,8.999999E+09,8.999999E+09,8.999999E+09,8.999999E+09,8.999999E+09]];
    LOCAL CONST Robtarget Tr_meulage_motif_1_126 := [[-313.67296875,-33.69679296875,12.7389482421875],[0.588012732058927,-0.500859688362471,0.411836559206125,-0.483498963816164],[0,0,0,0],[8.999999E+09,8.999999E+09,8.999999E+09,8.999999E+09,8.999999E+09,8.999999E+09]];
    LOCAL CONST Robtarget Tr_meulage_motif_1_127 := [[-313.44825,-34.67121484375,12.73948046875],[0.588012732058927,-0.500859688362471,0.411836559206125,-0.483498963816164],[0,0,0,0],[8.999999E+09,8.999999E+09,8.999999E+09,8.999999E+09,8.999999E+09,8.999999E+09]];
    LOCAL CONST Robtarget Tr_meulage_motif_1_128 := [[-313.22353125,-35.64563671875,12.7400126953125],[0.588012732058927,-0.500859688362471,0.411836559206125,-0.483498963816164],[0,0,0,0],[8.999999E+09,8.999999E+09,8.999999E+09,8.999999E+09,8.999999E+09,8.999999E+09]];
    LOCAL CONST Robtarget Tr_meulage_motif_1_129 := [[-312.9988125,-36.6200625,12.740544921875],[0.588012732058927,-0.500859688362471,0.411836559206125,-0.483498963816164],[0,0,0,0],[8.999999E+09,8.999999E+09,8.999999E+09,8.999999E+09,8.999999E+09,8.999999E+09]];
    LOCAL CONST Robtarget Tr_meulage_motif_1_130 := [[-312.77409375,-37.594484375,12.7410771484375],[0.588012732058927,-0.500859688362471,0.411836559206125,-0.483498963816164],[0,0,0,0],[8.999999E+09,8.999999E+09,8.999999E+09,8.999999E+09,8.999999E+09,8.999999E+09]];
    LOCAL CONST Robtarget Tr_meulage_motif_1_131 := [[-312.54934375,-38.56890625,12.741609375],[0.588012732058927,-0.500859688362471,0.411836559206125,-0.483498963816164],[0,0,0,0],[8.999999E+09,8.999999E+09,8.999999E+09,8.999999E+09,8.999999E+09,8.999999E+09]];
    LOCAL CONST Robtarget Tr_meulage_motif_1_132 := [[-312.324625,-39.543328125,12.7421416015625],[0.588012732058927,-0.500859688362471,0.411836559206125,-0.483498963816164],[0,0,0,0],[8.999999E+09,8.999999E+09,8.999999E+09,8.999999E+09,8.999999E+09,8.999999E+09]];
    LOCAL CONST Robtarget Tr_meulage_motif_1_133 := [[-312.09990625,-40.51775,12.742673828125],[0.588012732058927,-0.500859688362471,0.411836559206125,-0.483498963816164],[0,0,0,0],[8.999999E+09,8.999999E+09,8.999999E+09,8.999999E+09,8.999999E+09,8.999999E+09]];
    LOCAL CONST Robtarget Tr_meulage_motif_1_134 := [[-311.8751875,-41.492171875,12.7432060546875],[0.588012732058927,-0.500859688362471,0.411836559206125,-0.483498963816164],[0,0,0,0],[8.999999E+09,8.999999E+09,8.999999E+09,8.999999E+09,8.999999E+09,8.999999E+09]];
    LOCAL CONST Robtarget Tr_meulage_motif_1_135 := [[-311.65046875,-42.46659375,12.74373828125],[0.588012732058927,-0.500859688362471,0.411836559206125,-0.483498963816164],[0,0,0,0],[8.999999E+09,8.999999E+09,8.999999E+09,8.999999E+09,8.999999E+09,8.999999E+09]];
    LOCAL CONST Robtarget Tr_meulage_motif_1_136 := [[-311.42571875,-43.441015625,12.7442705078125],[0.588012732058927,-0.500859688362471,0.411836559206125,-0.483498963816164],[0,0,0,0],[8.999999E+09,8.999999E+09,8.999999E+09,8.999999E+09,8.999999E+09,8.999999E+09]];
    LOCAL CONST Robtarget Tr_meulage_motif_1_137 := [[-311.201,-44.4154375,12.744802734375],[0.588012732058927,-0.500859688362471,0.411836559206125,-0.483498963816164],[0,0,0,0],[8.999999E+09,8.999999E+09,8.999999E+09,8.999999E+09,8.999999E+09,8.999999E+09]];
    LOCAL CONST Robtarget Tr_meulage_motif_1_138 := [[-310.97928125,-45.3829765625,12.6347451171875],[0.588012732058927,-0.500859688362471,0.411836559206125,-0.483498963816164],[0,0,0,0],[8.999999E+09,8.999999E+09,8.999999E+09,8.999999E+09,8.999999E+09,8.999999E+09]];
    LOCAL CONST Robtarget Tr_meulage_motif_1_139 := [[-310.76909375,-46.3059609375,12.4240771484375],[0.588012732058927,-0.500859688362471,0.411836559206125,-0.483498963816164],[0,0,0,0],[8.999999E+09,8.999999E+09,8.999999E+09,8.999999E+09,8.999999E+09,8.999999E+09]];
    LOCAL CONST Robtarget Tr_meulage_motif_1_140 := [[-310.5806875,-47.137765625,12.1527080078125],[0.588012732058927,-0.500859688362471,0.411836559206125,-0.483498963816164],[0,0,0,0],[8.999999E+09,8.999999E+09,8.999999E+09,8.999999E+09,8.999999E+09,8.999999E+09]];
    LOCAL CONST Robtarget Tr_meulage_motif_1_141 := [[-310.4154375,-47.8694296875,11.8771904296875],[0.588012732058927,-0.500859688362471,0.411836559206125,-0.483498963816164],[0,0,0,0],[8.999999E+09,8.999999E+09,8.999999E+09,8.999999E+09,8.999999E+09,8.999999E+09]];
    LOCAL CONST Robtarget Tr_meulage_motif_1_142 := [[-310.17534375,-48.94435546875,11.26169921875],[0.588012732058927,-0.500859688362471,0.411836559206125,-0.483498963816164],[0,0,0,0],[8.999999E+09,8.999999E+09,8.999999E+09,8.999999E+09,8.999999E+09,8.999999E+09]];
    LOCAL CONST Robtarget Tr_meulage_motif_1_143 := [[-309.95534375,-49.94483203125,10.41465234375],[0.588012732058927,-0.500859688362471,0.411836559206125,-0.483498963816164],[0,0,0,0],[8.999999E+09,8.999999E+09,8.999999E+09,8.999999E+09,8.999999E+09,8.999999E+09]];
    LOCAL CONST Robtarget Tr_meulage_motif_1_144 := [[-309.77703125,-50.77417578125,9.391306640625],[0.588012732058927,-0.500859688362471,0.411836559206125,-0.483498963816164],[0,0,0,0],[8.999999E+09,8.999999E+09,8.999999E+09,8.999999E+09,8.999999E+09,8.999999E+09]];
    LOCAL CONST Robtarget Tr_meulage_motif_1_145 := [[-309.680625,-51.25351953125,8.2754638671875],[0.588012732058927,-0.500859688362471,0.411836559206125,-0.483498963816164],[0,0,0,0],[8.999999E+09,8.999999E+09,8.999999E+09,8.999999E+09,8.999999E+09,8.999999E+09]];
    LOCAL CONST Robtarget Tr_meulage_motif_1_146 := [[-309.68284375,-51.28218359375,7.5795625],[0.588012732058927,-0.500859688362471,0.411836559206125,-0.483498963816164],[0,0,0,0],[8.999999E+09,8.999999E+09,8.999999E+09,8.999999E+09,8.999999E+09,8.999999E+09]];
    LOCAL CONST Robtarget Tr_meulage_motif_1_147 := [[-309.69071875,-51.284359375,6.91836279296875],[0.588012732058927,-0.500859688362471,0.411836559206125,-0.483498963816164],[0,0,0,0],[8.999999E+09,8.999999E+09,8.999999E+09,8.999999E+09,8.999999E+09,8.999999E+09]];
    LOCAL CONST Robtarget Tr_meulage_motif_1_148 := [[-309.71090625,-51.2330625,6.2572900390625],[0.588012732058927,-0.500859688362471,0.411836559206125,-0.483498963816164],[0,0,0,0],[8.999999E+09,8.999999E+09,8.999999E+09,8.999999E+09,8.999999E+09,8.999999E+09]];
    LOCAL CONST Robtarget Tr_meulage_motif_1_149 := [[-309.836,-50.75121484375,5.155359375],[0.588012732058927,-0.500859688362471,0.411836559206125,-0.483498963816164],[0,0,0,0],[8.999999E+09,8.999999E+09,8.999999E+09,8.999999E+09,8.999999E+09,8.999999E+09]];
    LOCAL CONST Robtarget Tr_meulage_motif_1_150 := [[-310.04046875,-49.9198125,4.14835498046875],[0.588012732058927,-0.500859688362471,0.411836559206125,-0.483498963816164],[0,0,0,0],[8.999999E+09,8.999999E+09,8.999999E+09,8.999999E+09,8.999999E+09,8.999999E+09]];
    LOCAL CONST Robtarget Tr_meulage_motif_1_151 := [[-310.2803125,-48.9253125,3.31899877929688],[0.588012732058927,-0.500859688362471,0.411836559206125,-0.483498963816164],[0,0,0,0],[8.999999E+09,8.999999E+09,8.999999E+09,8.999999E+09,8.999999E+09,8.999999E+09]];
    LOCAL CONST Robtarget Tr_meulage_motif_1_152 := [[-310.4394375,-48.25709375,2.92291333007813],[0.588012732058927,-0.500859688362471,0.411836559206125,-0.483498963816164],[0,0,0,0],[8.999999E+09,8.999999E+09,8.999999E+09,8.999999E+09,8.999999E+09,8.999999E+09]];
    LOCAL CONST Robtarget Tr_meulage_motif_1_153 := [[-310.7055,-47.13016796875,2.43480297851562],[0.588012732058927,-0.500859688362471,0.411836559206125,-0.483498963816164],[0,0,0,0],[8.999999E+09,8.999999E+09,8.999999E+09,8.999999E+09,8.999999E+09,8.999999E+09]];
    LOCAL CONST Robtarget Tr_meulage_motif_1_154 := [[-310.8985625,-46.30762109375,2.17027954101563],[0.588012732058927,-0.500859688362471,0.411836559206125,-0.483498963816164],[0,0,0,0],[8.999999E+09,8.999999E+09,8.999999E+09,8.999999E+09,8.999999E+09,8.999999E+09]];
    LOCAL CONST Robtarget Tr_meulage_motif_1_155 := [[-311.1104375,-45.4001328125,1.96533056640625],[0.588012732058927,-0.500859688362471,0.411836559206125,-0.483498963816164],[0,0,0,0],[8.999999E+09,8.999999E+09,8.999999E+09,8.999999E+09,8.999999E+09,8.999999E+09]];
    LOCAL CONST Robtarget Tr_meulage_motif_1_156 := [[-311.3323125,-44.44403125,1.85622277832031],[0.588012732058927,-0.500859688362471,0.411836559206125,-0.483498963816164],[0,0,0,0],[8.999999E+09,8.999999E+09,8.999999E+09,8.999999E+09,8.999999E+09,8.999999E+09]];
    LOCAL CONST Robtarget Tr_meulage_motif_1_157 := [[-311.5566875,-43.47722265625,1.74510925292969],[0.588012732058927,-0.500859688362471,0.411836559206125,-0.483498963816164],[0,0,0,0],[8.999999E+09,8.999999E+09,8.999999E+09,8.999999E+09,8.999999E+09,8.999999E+09]];
    LOCAL CONST Robtarget Tr_meulage_motif_1_158 := [[-311.78140625,-42.50280078125,1.74457702636719],[0.588012732058927,-0.500859688362471,0.411836559206125,-0.483498963816164],[0,0,0,0],[8.999999E+09,8.999999E+09,8.999999E+09,8.999999E+09,8.999999E+09,8.999999E+09]];
    LOCAL CONST Robtarget Tr_meulage_motif_1_159 := [[-312.006125,-41.52837890625,1.744044921875],[0.588012732058927,-0.500859688362471,0.411836559206125,-0.483498963816164],[0,0,0,0],[8.999999E+09,8.999999E+09,8.999999E+09,8.999999E+09,8.999999E+09,8.999999E+09]];
    LOCAL CONST Robtarget Tr_meulage_motif_1_160 := [[-312.23084375,-40.55395703125,1.74351281738281],[0.588012732058927,-0.500859688362471,0.411836559206125,-0.483498963816164],[0,0,0,0],[8.999999E+09,8.999999E+09,8.999999E+09,8.999999E+09,8.999999E+09,8.999999E+09]];
    LOCAL CONST Robtarget Tr_meulage_motif_1_161 := [[-312.45559375,-39.57953515625,1.74298059082031],[0.588012732058927,-0.500859688362471,0.411836559206125,-0.483498963816164],[0,0,0,0],[8.999999E+09,8.999999E+09,8.999999E+09,8.999999E+09,8.999999E+09,8.999999E+09]];
    LOCAL CONST Robtarget Tr_meulage_motif_1_162 := [[-312.6803125,-38.60511328125,1.74244848632813],[0.588012732058927,-0.500859688362471,0.411836559206125,-0.483498963816164],[0,0,0,0],[8.999999E+09,8.999999E+09,8.999999E+09,8.999999E+09,8.999999E+09,8.999999E+09]];
    LOCAL CONST Robtarget Tr_meulage_motif_1_163 := [[-312.90503125,-37.6306875,1.74191638183594],[0.588012732058927,-0.500859688362471,0.411836559206125,-0.483498963816164],[0,0,0,0],[8.999999E+09,8.999999E+09,8.999999E+09,8.999999E+09,8.999999E+09,8.999999E+09]];
    LOCAL CONST Robtarget Tr_meulage_motif_1_164 := [[-313.12975,-36.656265625,1.74138415527344],[0.588012732058927,-0.500859688362471,0.411836559206125,-0.483498963816164],[0,0,0,0],[8.999999E+09,8.999999E+09,8.999999E+09,8.999999E+09,8.999999E+09,8.999999E+09]];
    LOCAL CONST Robtarget Tr_meulage_motif_1_165 := [[-313.35446875,-35.68184375,1.74085205078125],[0.588012732058927,-0.500859688362471,0.411836559206125,-0.483498963816164],[0,0,0,0],[8.999999E+09,8.999999E+09,8.999999E+09,8.999999E+09,8.999999E+09,8.999999E+09]];
    LOCAL CONST Robtarget Tr_meulage_motif_1_166 := [[-313.57921875,-34.707421875,1.74031994628906],[0.588012732058927,-0.500859688362471,0.411836559206125,-0.483498963816164],[0,0,0,0],[8.999999E+09,8.999999E+09,8.999999E+09,8.999999E+09,8.999999E+09,8.999999E+09]];
    LOCAL CONST Robtarget Tr_meulage_motif_1_167 := [[-313.8039375,-33.733,1.73978771972656],[0.588012732058927,-0.500859688362471,0.411836559206125,-0.483498963816164],[0,0,0,0],[8.999999E+09,8.999999E+09,8.999999E+09,8.999999E+09,8.999999E+09,8.999999E+09]];
    LOCAL CONST Robtarget Tr_meulage_motif_1_168 := [[-314.02865625,-32.758578125,1.73925561523437],[0.588012732058927,-0.500859688362471,0.411836559206125,-0.483498963816164],[0,0,0,0],[8.999999E+09,8.999999E+09,8.999999E+09,8.999999E+09,8.999999E+09,8.999999E+09]];
    LOCAL CONST Robtarget Tr_meulage_motif_1_169 := [[-314.253375,-31.78415625,1.73872351074219],[0.588012732058927,-0.500859688362471,0.411836559206125,-0.483498963816164],[0,0,0,0],[8.999999E+09,8.999999E+09,8.999999E+09,8.999999E+09,8.999999E+09,8.999999E+09]];
    LOCAL CONST Robtarget Tr_meulage_motif_1_170 := [[-314.47809375,-30.809734375,1.73819128417969],[0.588012732058927,-0.500859688362471,0.411836559206125,-0.483498963816164],[0,0,0,0],[8.999999E+09,8.999999E+09,8.999999E+09,8.999999E+09,8.999999E+09,8.999999E+09]];
    LOCAL CONST Robtarget Tr_meulage_motif_1_171 := [[-314.70284375,-29.8353125,1.7376591796875],[0.588012732058927,-0.500859688362471,0.411836559206125,-0.483498963816164],[0,0,0,0],[8.999999E+09,8.999999E+09,8.999999E+09,8.999999E+09,8.999999E+09,8.999999E+09]];
    LOCAL CONST Robtarget Tr_meulage_motif_1_172 := [[-314.9275625,-28.860890625,1.73712707519531],[0.588012732058927,-0.500859688362471,0.411836559206125,-0.483498963816164],[0,0,0,0],[8.999999E+09,8.999999E+09,8.999999E+09,8.999999E+09,8.999999E+09,8.999999E+09]];
    LOCAL CONST Robtarget Tr_meulage_motif_1_173 := [[-315.15228125,-27.88646875,1.73659484863281],[0.588012732058927,-0.500859688362471,0.411836559206125,-0.483498963816164],[0,0,0,0],[8.999999E+09,8.999999E+09,8.999999E+09,8.999999E+09,8.999999E+09,8.999999E+09]];
    LOCAL CONST Robtarget Tr_meulage_motif_1_174 := [[-315.377,-26.912046875,1.73606274414063],[0.588012732058927,-0.500859688362471,0.411836559206125,-0.483498963816164],[0,0,0,0],[8.999999E+09,8.999999E+09,8.999999E+09,8.999999E+09,8.999999E+09,8.999999E+09]];
    LOCAL CONST Robtarget Tr_meulage_motif_1_175 := [[-315.60171875,-25.937625,1.73553063964844],[0.588012732058927,-0.500859688362471,0.411836559206125,-0.483498963816164],[0,0,0,0],[8.999999E+09,8.999999E+09,8.999999E+09,8.999999E+09,8.999999E+09,8.999999E+09]];
    LOCAL CONST Robtarget Tr_meulage_motif_1_176 := [[-315.82646875,-24.963203125,1.73499841308594],[0.588012732058927,-0.500859688362471,0.411836559206125,-0.483498963816164],[0,0,0,0],[8.999999E+09,8.999999E+09,8.999999E+09,8.999999E+09,8.999999E+09,8.999999E+09]];
    LOCAL CONST Robtarget Tr_meulage_motif_1_177 := [[-316.0511875,-23.98878125,1.73446630859375],[0.588012732058927,-0.500859688362471,0.411836559206125,-0.483498963816164],[0,0,0,0],[8.999999E+09,8.999999E+09,8.999999E+09,8.999999E+09,8.999999E+09,8.999999E+09]];
    LOCAL CONST Robtarget Tr_meulage_motif_1_178 := [[-316.27590625,-23.014359375,1.73393420410156],[0.588012732058927,-0.500859688362471,0.411836559206125,-0.483498963816164],[0,0,0,0],[8.999999E+09,8.999999E+09,8.999999E+09,8.999999E+09,8.999999E+09,8.999999E+09]];
    LOCAL CONST Robtarget Tr_meulage_motif_1_179 := [[-316.500625,-22.039935546875,1.73340197753906],[0.588012732058927,-0.500859688362471,0.411836559206125,-0.483498963816164],[0,0,0,0],[8.999999E+09,8.999999E+09,8.999999E+09,8.999999E+09,8.999999E+09,8.999999E+09]];
    LOCAL CONST Robtarget Tr_meulage_motif_1_180 := [[-316.72534375,-21.065513671875,1.73286987304688],[0.588012732058927,-0.500859688362471,0.411836559206125,-0.483498963816164],[0,0,0,0],[8.999999E+09,8.999999E+09,8.999999E+09,8.999999E+09,8.999999E+09,8.999999E+09]];
    LOCAL CONST Robtarget Tr_meulage_motif_1_181 := [[-316.95009375,-20.091091796875,1.73233776855469],[0.588012732058927,-0.500859688362471,0.411836559206125,-0.483498963816164],[0,0,0,0],[8.999999E+09,8.999999E+09,8.999999E+09,8.999999E+09,8.999999E+09,8.999999E+09]];
    LOCAL CONST Robtarget Tr_meulage_motif_1_182 := [[-317.1748125,-19.116669921875,1.73180554199219],[0.588012732058927,-0.500859688362471,0.411836559206125,-0.483498963816164],[0,0,0,0],[8.999999E+09,8.999999E+09,8.999999E+09,8.999999E+09,8.999999E+09,8.999999E+09]];
    LOCAL CONST Robtarget Tr_meulage_motif_1_183 := [[-317.39953125,-18.142248046875,1.7312734375],[0.588012732058927,-0.500859688362471,0.411836559206125,-0.483498963816164],[0,0,0,0],[8.999999E+09,8.999999E+09,8.999999E+09,8.999999E+09,8.999999E+09,8.999999E+09]];
    LOCAL CONST Robtarget Tr_meulage_motif_1_184 := [[-317.62425,-17.167826171875,1.73074133300781],[0.588012732058927,-0.500859688362471,0.411836559206125,-0.483498963816164],[0,0,0,0],[8.999999E+09,8.999999E+09,8.999999E+09,8.999999E+09,8.999999E+09,8.999999E+09]];
    LOCAL CONST Robtarget Tr_meulage_motif_1_185 := [[-317.84896875,-16.193404296875,1.73020910644531],[0.588012732058927,-0.500859688362471,0.411836559206125,-0.483498963816164],[0,0,0,0],[8.999999E+09,8.999999E+09,8.999999E+09,8.999999E+09,8.999999E+09,8.999999E+09]];
    LOCAL CONST Robtarget Tr_meulage_motif_1_186 := [[-318.07371875,-15.2189814453125,1.72967700195313],[0.588012732058927,-0.500859688362471,0.411836559206125,-0.483498963816164],[0,0,0,0],[8.999999E+09,8.999999E+09,8.999999E+09,8.999999E+09,8.999999E+09,8.999999E+09]];
    LOCAL CONST Robtarget Tr_meulage_motif_1_187 := [[-318.2984375,-14.2445595703125,1.72914489746094],[0.588012732058927,-0.500859688362471,0.411836559206125,-0.483498963816164],[0,0,0,0],[8.999999E+09,8.999999E+09,8.999999E+09,8.999999E+09,8.999999E+09,8.999999E+09]];
    LOCAL CONST Robtarget Tr_meulage_motif_1_188 := [[-318.5228125,-13.2777490234375,1.61803137207031],[0.588012732058927,-0.500859688362471,0.411836559206125,-0.483498963816164],[0,0,0,0],[8.999999E+09,8.999999E+09,8.999999E+09,8.999999E+09,8.999999E+09,8.999999E+09]];
    LOCAL CONST Robtarget Tr_meulage_motif_1_189 := [[-318.73803125,-12.3561533203125,1.40635632324219],[0.588012732058927,-0.500859688362471,0.411836559206125,-0.483498963816164],[0,0,0,0],[8.999999E+09,8.999999E+09,8.999999E+09,8.999999E+09,8.999999E+09,8.999999E+09]];
    LOCAL CONST Robtarget Tr_meulage_motif_1_190 := [[-318.932875,-11.526140625,1.13407946777344],[0.588012732058927,-0.500859688362471,0.411836559206125,-0.483498963816164],[0,0,0,0],[8.999999E+09,8.999999E+09,8.999999E+09,8.999999E+09,8.999999E+09,8.999999E+09]];
    LOCAL CONST Robtarget Tr_meulage_motif_1_191 := [[-319.09640625,-10.83383984375,0.82958349609375],[0.588012732058927,-0.500859688362471,0.411836559206125,-0.483498963816164],[0,0,0,0],[8.999999E+09,8.999999E+09,8.999999E+09,8.999999E+09,8.999999E+09,8.999999E+09]];
    LOCAL CONST Robtarget Tr_meulage_motif_1_192 := [[-319.33675,-9.82801171875,0.166552261352539],[0.588012732058927,-0.500859688362471,0.411836559206125,-0.483498963816164],[0,0,0,0],[8.999999E+09,8.999999E+09,8.999999E+09,8.999999E+09,8.999999E+09,8.999999E+09]];
    LOCAL CONST Robtarget Tr_meulage_motif_1_193 := [[-319.5501875,-8.95211328125,-0.73581201171875],[0.588012732058927,-0.500859688362471,0.411836559206125,-0.483498963816164],[0,0,0,0],[8.999999E+09,8.999999E+09,8.999999E+09,8.999999E+09,8.999999E+09,8.999999E+09]];
    LOCAL CONST Robtarget Tr_meulage_motif_1_194 := [[-319.68284375,-8.4342705078125,-1.78203259277344],[0.588012732058927,-0.500859688362471,0.411836559206125,-0.483498963816164],[0,0,0,0],[8.999999E+09,8.999999E+09,8.999999E+09,8.999999E+09,8.999999E+09,8.999999E+09]];
    LOCAL CONST Robtarget Tr_meulage_motif_1_195 := [[-319.732625,-8.2564970703125,-2.47531225585938],[0.588012732058927,-0.500859688362471,0.411836559206125,-0.483498963816164],[0,0,0,0],[8.999999E+09,8.999999E+09,8.999999E+09,8.999999E+09,8.999999E+09,8.999999E+09]];
    LOCAL CONST Robtarget Tr_meulage_motif_1_196 := [[-319.75615625,-8.1968212890625,-3.24528759765625],[0.588012732058927,-0.500859688362471,0.411836559206125,-0.483498963816164],[0,0,0,0],[8.999999E+09,8.999999E+09,8.999999E+09,8.999999E+09,8.999999E+09,8.999999E+09]];
    LOCAL CONST Robtarget Tr_meulage_motif_1_197 := [[-319.75028125,-8.264580078125,-4.015052734375],[0.588012732058927,-0.500859688362471,0.411836559206125,-0.483498963816164],[0,0,0,0],[8.999999E+09,8.999999E+09,8.999999E+09,8.999999E+09,8.999999E+09,8.999999E+09]];
    LOCAL CONST Robtarget Tr_meulage_motif_1_198 := [[-319.66915625,-8.67708984375,-5.12299462890625],[0.588012732058927,-0.500859688362471,0.411836559206125,-0.483498963816164],[0,0,0,0],[8.999999E+09,8.999999E+09,8.999999E+09,8.999999E+09,8.999999E+09,8.999999E+09]];
    LOCAL CONST Robtarget Tr_meulage_motif_1_199 := [[-319.58303125,-9.082732421875,-5.7084169921875],[0.588012732058927,-0.500859688362471,0.411836559206125,-0.483498963816164],[0,0,0,0],[8.999999E+09,8.999999E+09,8.999999E+09,8.999999E+09,8.999999E+09,8.999999E+09]];
    LOCAL CONST Robtarget Tr_meulage_motif_1_200 := [[-319.39421875,-9.9500869140625,-6.59503369140625],[0.588012732058927,-0.500859688362471,0.411836559206125,-0.483498963816164],[0,0,0,0],[8.999999E+09,8.999999E+09,8.999999E+09,8.999999E+09,8.999999E+09,8.999999E+09]];
    LOCAL CONST Robtarget Tr_meulage_motif_1_201 := [[-319.26753125,-10.5221572265625,-7.0089716796875],[0.588012732058927,-0.500859688362471,0.411836559206125,-0.483498963816164],[0,0,0,0],[8.999999E+09,8.999999E+09,8.999999E+09,8.999999E+09,8.999999E+09,8.999999E+09]];
    LOCAL CONST Robtarget Tr_meulage_motif_1_202 := [[-319.0228125,-11.6132607421875,-7.55246044921875],[0.588012732058927,-0.500859688362471,0.411836559206125,-0.483498963816164],[0,0,0,0],[8.999999E+09,8.999999E+09,8.999999E+09,8.999999E+09,8.999999E+09,8.999999E+09]];
    LOCAL CONST Robtarget Tr_meulage_motif_1_203 := [[-318.84078125,-12.4187099609375,-7.84749853515625],[0.588012732058927,-0.500859688362471,0.411836559206125,-0.483498963816164],[0,0,0,0],[8.999999E+09,8.999999E+09,8.999999E+09,8.999999E+09,8.999999E+09,8.999999E+09]];
    LOCAL CONST Robtarget Tr_meulage_motif_1_204 := [[-318.63378125,-13.327544921875,-8.05147119140625],[0.588012732058927,-0.500859688362471,0.411836559206125,-0.483498963816164],[0,0,0,0],[8.999999E+09,8.999999E+09,8.999999E+09,8.999999E+09,8.999999E+09,8.999999E+09]];
    LOCAL CONST Robtarget Tr_meulage_motif_1_205 := [[-318.4145,-14.2843583984375,-8.1594873046875],[0.588012732058927,-0.500859688362471,0.411836559206125,-0.483498963816164],[0,0,0,0],[8.999999E+09,8.999999E+09,8.999999E+09,8.999999E+09,8.999999E+09,8.999999E+09]];
    LOCAL CONST Robtarget Tr_meulage_motif_1_206 := [[-318.19275,-15.2518974609375,-8.269560546875],[0.588012732058927,-0.500859688362471,0.411836559206125,-0.483498963816164],[0,0,0,0],[8.999999E+09,8.999999E+09,8.999999E+09,8.999999E+09,8.999999E+09,8.999999E+09]];
    LOCAL CONST Robtarget Tr_meulage_motif_1_207 := [[-317.96803125,-16.2263193359375,-8.2690283203125],[0.588012732058927,-0.500859688362471,0.411836559206125,-0.483498963816164],[0,0,0,0],[8.999999E+09,8.999999E+09,8.999999E+09,8.999999E+09,8.999999E+09,8.999999E+09]];
    LOCAL CONST Robtarget Tr_meulage_motif_1_208 := [[-317.7433125,-17.200740234375,-8.26849609375],[0.588012732058927,-0.500859688362471,0.411836559206125,-0.483498963816164],[0,0,0,0],[8.999999E+09,8.999999E+09,8.999999E+09,8.999999E+09,8.999999E+09,8.999999E+09]];
    LOCAL CONST Robtarget Tr_meulage_motif_1_209 := [[-317.5185625,-18.1751640625,-8.2679638671875],[0.588012732058927,-0.500859688362471,0.411836559206125,-0.483498963816164],[0,0,0,0],[8.999999E+09,8.999999E+09,8.999999E+09,8.999999E+09,8.999999E+09,8.999999E+09]];
    LOCAL CONST Robtarget Tr_meulage_motif_1_210 := [[-317.29384375,-19.1495859375,-8.267431640625],[0.588012732058927,-0.500859688362471,0.411836559206125,-0.483498963816164],[0,0,0,0],[8.999999E+09,8.999999E+09,8.999999E+09,8.999999E+09,8.999999E+09,8.999999E+09]];
    LOCAL CONST Robtarget Tr_meulage_motif_1_211 := [[-317.069125,-20.1240078125,-8.2668994140625],[0.588012732058927,-0.500859688362471,0.411836559206125,-0.483498963816164],[0,0,0,0],[8.999999E+09,8.999999E+09,8.999999E+09,8.999999E+09,8.999999E+09,8.999999E+09]];
    LOCAL CONST Robtarget Tr_meulage_motif_1_212 := [[-316.84440625,-21.0984296875,-8.2663671875],[0.588012732058927,-0.500859688362471,0.411836559206125,-0.483498963816164],[0,0,0,0],[8.999999E+09,8.999999E+09,8.999999E+09,8.999999E+09,8.999999E+09,8.999999E+09]];
    LOCAL CONST Robtarget Tr_meulage_motif_1_213 := [[-316.6196875,-22.0728515625,-8.2658349609375],[0.588012732058927,-0.500859688362471,0.411836559206125,-0.483498963816164],[0,0,0,0],[8.999999E+09,8.999999E+09,8.999999E+09,8.999999E+09,8.999999E+09,8.999999E+09]];
    LOCAL CONST Robtarget Tr_meulage_motif_1_214 := [[-316.3949375,-23.0472734375,-8.265302734375],[0.588012732058927,-0.500859688362471,0.411836559206125,-0.483498963816164],[0,0,0,0],[8.999999E+09,8.999999E+09,8.999999E+09,8.999999E+09,8.999999E+09,8.999999E+09]];
    LOCAL CONST Robtarget Tr_meulage_motif_1_215 := [[-316.17021875,-24.0216953125,-8.2647705078125],[0.588012732058927,-0.500859688362471,0.411836559206125,-0.483498963816164],[0,0,0,0],[8.999999E+09,8.999999E+09,8.999999E+09,8.999999E+09,8.999999E+09,8.999999E+09]];
    LOCAL CONST Robtarget Tr_meulage_motif_1_216 := [[-315.9455,-24.9961171875,-8.26423828125],[0.588012732058927,-0.500859688362471,0.411836559206125,-0.483498963816164],[0,0,0,0],[8.999999E+09,8.999999E+09,8.999999E+09,8.999999E+09,8.999999E+09,8.999999E+09]];
    LOCAL CONST Robtarget Tr_meulage_motif_1_217 := [[-315.72078125,-25.9705390625,-8.26370703125],[0.588012732058927,-0.500859688362471,0.411836559206125,-0.483498963816164],[0,0,0,0],[8.999999E+09,8.999999E+09,8.999999E+09,8.999999E+09,8.999999E+09,8.999999E+09]];
    LOCAL CONST Robtarget Tr_meulage_motif_1_218 := [[-315.4960625,-26.9449609375,-8.2631748046875],[0.588012732058927,-0.500859688362471,0.411836559206125,-0.483498963816164],[0,0,0,0],[8.999999E+09,8.999999E+09,8.999999E+09,8.999999E+09,8.999999E+09,8.999999E+09]];
    LOCAL CONST Robtarget Tr_meulage_motif_1_219 := [[-315.2713125,-27.919384765625,-8.262642578125],[0.588012732058927,-0.500859688362471,0.411836559206125,-0.483498963816164],[0,0,0,0],[8.999999E+09,8.999999E+09,8.999999E+09,8.999999E+09,8.999999E+09,8.999999E+09]];
    LOCAL CONST Robtarget Tr_meulage_motif_1_220 := [[-315.04659375,-28.893806640625,-8.2621103515625],[0.588012732058927,-0.500859688362471,0.411836559206125,-0.483498963816164],[0,0,0,0],[8.999999E+09,8.999999E+09,8.999999E+09,8.999999E+09,8.999999E+09,8.999999E+09]];
    LOCAL CONST Robtarget Tr_meulage_motif_1_221 := [[-314.821875,-29.868228515625,-8.261578125],[0.588012732058927,-0.500859688362471,0.411836559206125,-0.483498963816164],[0,0,0,0],[8.999999E+09,8.999999E+09,8.999999E+09,8.999999E+09,8.999999E+09,8.999999E+09]];
    LOCAL CONST Robtarget Tr_meulage_motif_1_222 := [[-314.59715625,-30.842650390625,-8.2610458984375],[0.588012732058927,-0.500859688362471,0.411836559206125,-0.483498963816164],[0,0,0,0],[8.999999E+09,8.999999E+09,8.999999E+09,8.999999E+09,8.999999E+09,8.999999E+09]];
    LOCAL CONST Robtarget Tr_meulage_motif_1_223 := [[-314.3724375,-31.817072265625,-8.260513671875],[0.588012732058927,-0.500859688362471,0.411836559206125,-0.483498963816164],[0,0,0,0],[8.999999E+09,8.999999E+09,8.999999E+09,8.999999E+09,8.999999E+09,8.999999E+09]];
    LOCAL CONST Robtarget Tr_meulage_motif_1_224 := [[-314.1476875,-32.79149609375,-8.2599814453125],[0.588012732058927,-0.500859688362471,0.411836559206125,-0.483498963816164],[0,0,0,0],[8.999999E+09,8.999999E+09,8.999999E+09,8.999999E+09,8.999999E+09,8.999999E+09]];
    LOCAL CONST Robtarget Tr_meulage_motif_1_225 := [[-313.92296875,-33.76591796875,-8.25944921875],[0.588012732058927,-0.500859688362471,0.411836559206125,-0.483498963816164],[0,0,0,0],[8.999999E+09,8.999999E+09,8.999999E+09,8.999999E+09,8.999999E+09,8.999999E+09]];
    LOCAL CONST Robtarget Tr_meulage_motif_1_226 := [[-313.69825,-34.74033984375,-8.2589169921875],[0.588012732058927,-0.500859688362471,0.411836559206125,-0.483498963816164],[0,0,0,0],[8.999999E+09,8.999999E+09,8.999999E+09,8.999999E+09,8.999999E+09,8.999999E+09]];
    LOCAL CONST Robtarget Tr_meulage_motif_1_227 := [[-313.47353125,-35.71476171875,-8.258384765625],[0.588012732058927,-0.500859688362471,0.411836559206125,-0.483498963816164],[0,0,0,0],[8.999999E+09,8.999999E+09,8.999999E+09,8.999999E+09,8.999999E+09,8.999999E+09]];
    LOCAL CONST Robtarget Tr_meulage_motif_1_228 := [[-313.2488125,-36.68918359375,-8.2578525390625],[0.588012732058927,-0.500859688362471,0.411836559206125,-0.483498963816164],[0,0,0,0],[8.999999E+09,8.999999E+09,8.999999E+09,8.999999E+09,8.999999E+09,8.999999E+09]];
    LOCAL CONST Robtarget Tr_meulage_motif_1_229 := [[-313.0240625,-37.66360546875,-8.2573212890625],[0.588012732058927,-0.500859688362471,0.411836559206125,-0.483498963816164],[0,0,0,0],[8.999999E+09,8.999999E+09,8.999999E+09,8.999999E+09,8.999999E+09,8.999999E+09]];
    LOCAL CONST Robtarget Tr_meulage_motif_1_230 := [[-312.79934375,-38.63802734375,-8.2567890625],[0.588012732058927,-0.500859688362471,0.411836559206125,-0.483498963816164],[0,0,0,0],[8.999999E+09,8.999999E+09,8.999999E+09,8.999999E+09,8.999999E+09,8.999999E+09]];
    LOCAL CONST Robtarget Tr_meulage_motif_1_231 := [[-312.574625,-39.61244921875,-8.2562568359375],[0.588012732058927,-0.500859688362471,0.411836559206125,-0.483498963816164],[0,0,0,0],[8.999999E+09,8.999999E+09,8.999999E+09,8.999999E+09,8.999999E+09,8.999999E+09]];
    LOCAL CONST Robtarget Tr_meulage_motif_1_232 := [[-312.34990625,-40.58687109375,-8.255724609375],[0.588012732058927,-0.500859688362471,0.411836559206125,-0.483498963816164],[0,0,0,0],[8.999999E+09,8.999999E+09,8.999999E+09,8.999999E+09,8.999999E+09,8.999999E+09]];
    LOCAL CONST Robtarget Tr_meulage_motif_1_233 := [[-312.1251875,-41.56129296875,-8.2551923828125],[0.588012732058927,-0.500859688362471,0.411836559206125,-0.483498963816164],[0,0,0,0],[8.999999E+09,8.999999E+09,8.999999E+09,8.999999E+09,8.999999E+09,8.999999E+09]];
    LOCAL CONST Robtarget Tr_meulage_motif_1_234 := [[-311.9004375,-42.53571484375,-8.25466015625],[0.588012732058927,-0.500859688362471,0.411836559206125,-0.483498963816164],[0,0,0,0],[8.999999E+09,8.999999E+09,8.999999E+09,8.999999E+09,8.999999E+09,8.999999E+09]];
    LOCAL CONST Robtarget Tr_meulage_motif_1_235 := [[-311.67571875,-43.51013671875,-8.2541279296875],[0.588012732058927,-0.500859688362471,0.411836559206125,-0.483498963816164],[0,0,0,0],[8.999999E+09,8.999999E+09,8.999999E+09,8.999999E+09,8.999999E+09,8.999999E+09]];
    LOCAL CONST Robtarget Tr_meulage_motif_1_236 := [[-311.451,-44.48455859375,-8.253595703125],[0.588012732058927,-0.500859688362471,0.411836559206125,-0.483498963816164],[0,0,0,0],[8.999999E+09,8.999999E+09,8.999999E+09,8.999999E+09,8.999999E+09,8.999999E+09]];
    LOCAL CONST Robtarget Tr_meulage_motif_1_237 := [[-311.22925,-45.45209765625,-8.3636689453125],[0.588012732058927,-0.500859688362471,0.411836559206125,-0.483498963816164],[0,0,0,0],[8.999999E+09,8.999999E+09,8.999999E+09,8.999999E+09,8.999999E+09,8.999999E+09]];
    LOCAL CONST Robtarget Tr_meulage_motif_1_238 := [[-311.0190625,-46.37508203125,-8.5743359375],[0.588012732058927,-0.500859688362471,0.411836559206125,-0.483498963816164],[0,0,0,0],[8.999999E+09,8.999999E+09,8.999999E+09,8.999999E+09,8.999999E+09,8.999999E+09]];
    LOCAL CONST Robtarget Tr_meulage_motif_1_239 := [[-310.8306875,-47.20688671875,-8.8456904296875],[0.588012732058927,-0.500859688362471,0.411836559206125,-0.483498963816164],[0,0,0,0],[8.999999E+09,8.999999E+09,8.999999E+09,8.999999E+09,8.999999E+09,8.999999E+09]];
    LOCAL CONST Robtarget Tr_meulage_motif_1_240 := [[-310.67440625,-47.9011875,-9.1494287109375],[0.588012732058927,-0.500859688362471,0.411836559206125,-0.483498963816164],[0,0,0,0],[8.999999E+09,8.999999E+09,8.999999E+09,8.999999E+09,8.999999E+09,8.999999E+09]];
    LOCAL CONST Robtarget Tr_meulage_motif_1_241 := [[-310.44984375,-48.91137890625,-9.811359375],[0.588012732058927,-0.500859688362471,0.411836559206125,-0.483498963816164],[0,0,0,0],[8.999999E+09,8.999999E+09,8.999999E+09,8.999999E+09,8.999999E+09,8.999999E+09]];
    LOCAL CONST Robtarget Tr_meulage_motif_1_242 := [[-310.27834375,-49.7065546875,-10.7506357421875],[0.588012732058927,-0.500859688362471,0.411836559206125,-0.483498963816164],[0,0,0,0],[8.999999E+09,8.999999E+09,8.999999E+09,8.999999E+09,8.999999E+09,8.999999E+09]];
    LOCAL CONST Robtarget Tr_meulage_motif_1_243 := [[-310.211,-50.0532578125,-11.7467314453125],[0.588012732058927,-0.500859688362471,0.411836559206125,-0.483498963816164],[0,0,0,0],[8.999999E+09,8.999999E+09,8.999999E+09,8.999999E+09,8.999999E+09,8.999999E+09]];
    LOCAL CONST Robtarget Tr_meulage_motif_1_244 := [[-310.2243125,-50.0261953125,-12.304251953125],[0.588012732058927,-0.500859688362471,0.411836559206125,-0.483498963816164],[0,0,0,0],[8.999999E+09,8.999999E+09,8.999999E+09,8.999999E+09,8.999999E+09,8.999999E+09]];
    LOCAL CONST Robtarget Tr_meulage_motif_1_245 := [[-310.2283125,-50.0317734375,-12.7221240234375],[0.588012732058927,-0.500859688362471,0.411836559206125,-0.483498963816164],[0,0,0,0],[8.999999E+09,8.999999E+09,8.999999E+09,8.999999E+09,8.999999E+09,8.999999E+09]];
    LOCAL CONST Robtarget Tr_meulage_motif_1_246 := [[-310.32125,-49.6820703125,-13.6915712890625],[0.588012732058927,-0.500859688362471,0.411836559206125,-0.483498963816164],[0,0,0,0],[8.999999E+09,8.999999E+09,8.999999E+09,8.999999E+09,8.999999E+09,8.999999E+09]];
    LOCAL CONST Robtarget Tr_meulage_motif_1_247 := [[-310.516875,-48.88417578125,-14.6096259765625],[0.588012732058927,-0.500859688362471,0.411836559206125,-0.483498963816164],[0,0,0,0],[8.999999E+09,8.999999E+09,8.999999E+09,8.999999E+09,8.999999E+09,8.999999E+09]];
    LOCAL CONST Robtarget Tr_meulage_motif_1_248 := [[-310.65946875,-48.2890703125,-15.0328095703125],[0.588012732058927,-0.500859688362471,0.411836559206125,-0.483498963816164],[0,0,0,0],[8.999999E+09,8.999999E+09,8.999999E+09,8.999999E+09,8.999999E+09,8.999999E+09]];
    LOCAL CONST Robtarget Tr_meulage_motif_1_249 := [[-310.91978125,-47.1894140625,-15.56382421875],[0.588012732058927,-0.500859688362471,0.411836559206125,-0.483498963816164],[0,0,0,0],[8.999999E+09,8.999999E+09,8.999999E+09,8.999999E+09,8.999999E+09,8.999999E+09]];
    LOCAL CONST Robtarget Tr_meulage_motif_1_250 := [[-311.11284375,-46.3668671875,-15.82836328125],[0.588012732058927,-0.500859688362471,0.411836559206125,-0.483498963816164],[0,0,0,0],[8.999999E+09,8.999999E+09,8.999999E+09,8.999999E+09,8.999999E+09,8.999999E+09]];
    LOCAL CONST Robtarget Tr_meulage_motif_1_251 := [[-311.32471875,-45.45937890625,-16.033328125],[0.588012732058927,-0.500859688362471,0.411836559206125,-0.483498963816164],[0,0,0,0],[8.999999E+09,8.999999E+09,8.999999E+09,8.999999E+09,8.999999E+09,8.999999E+09]];
    LOCAL CONST Robtarget Tr_meulage_motif_1_252 := [[-311.54659375,-44.50328125,-16.142388671875],[0.588012732058927,-0.500859688362471,0.411836559206125,-0.483498963816164],[0,0,0,0],[8.999999E+09,8.999999E+09,8.999999E+09,8.999999E+09,8.999999E+09,8.999999E+09]];
    LOCAL CONST Robtarget Tr_meulage_motif_1_253 := [[-311.77096875,-43.53646875,-16.253517578125],[0.588012732058927,-0.500859688362471,0.411836559206125,-0.483498963816164],[0,0,0,0],[8.999999E+09,8.999999E+09,8.999999E+09,8.999999E+09,8.999999E+09,8.999999E+09]];
    LOCAL CONST Robtarget Tr_meulage_motif_1_254 := [[-311.9956875,-42.562046875,-16.2540498046875],[0.588012732058927,-0.500859688362471,0.411836559206125,-0.483498963816164],[0,0,0,0],[8.999999E+09,8.999999E+09,8.999999E+09,8.999999E+09,8.999999E+09,8.999999E+09]];
    LOCAL CONST Robtarget Tr_meulage_motif_1_255 := [[-312.22040625,-41.587625,-16.25458203125],[0.588012732058927,-0.500859688362471,0.411836559206125,-0.483498963816164],[0,0,0,0],[8.999999E+09,8.999999E+09,8.999999E+09,8.999999E+09,8.999999E+09,8.999999E+09]];
    LOCAL CONST Robtarget Tr_meulage_motif_1_256 := [[-312.445125,-40.613203125,-16.2551142578125],[0.588012732058927,-0.500859688362471,0.411836559206125,-0.483498963816164],[0,0,0,0],[8.999999E+09,8.999999E+09,8.999999E+09,8.999999E+09,8.999999E+09,8.999999E+09]];
    LOCAL CONST Robtarget Tr_meulage_motif_1_257 := [[-312.669875,-39.63878125,-16.255646484375],[0.588012732058927,-0.500859688362471,0.411836559206125,-0.483498963816164],[0,0,0,0],[8.999999E+09,8.999999E+09,8.999999E+09,8.999999E+09,8.999999E+09,8.999999E+09]];
    LOCAL CONST Robtarget Tr_meulage_motif_1_258 := [[-312.89459375,-38.664359375,-16.2561787109375],[0.588012732058927,-0.500859688362471,0.411836559206125,-0.483498963816164],[0,0,0,0],[8.999999E+09,8.999999E+09,8.999999E+09,8.999999E+09,8.999999E+09,8.999999E+09]];
    LOCAL CONST Robtarget Tr_meulage_motif_1_259 := [[-313.1193125,-37.6899375,-16.2567109375],[0.588012732058927,-0.500859688362471,0.411836559206125,-0.483498963816164],[0,0,0,0],[8.999999E+09,8.999999E+09,8.999999E+09,8.999999E+09,8.999999E+09,8.999999E+09]];
    LOCAL CONST Robtarget Tr_meulage_motif_1_260 := [[-313.34403125,-36.715515625,-16.2572431640625],[0.588012732058927,-0.500859688362471,0.411836559206125,-0.483498963816164],[0,0,0,0],[8.999999E+09,8.999999E+09,8.999999E+09,8.999999E+09,8.999999E+09,8.999999E+09]];
    LOCAL CONST Robtarget Tr_meulage_motif_1_261 := [[-313.56875,-35.74109375,-16.257775390625],[0.588012732058927,-0.500859688362471,0.411836559206125,-0.483498963816164],[0,0,0,0],[8.999999E+09,8.999999E+09,8.999999E+09,8.999999E+09,8.999999E+09,8.999999E+09]];
    LOCAL CONST Robtarget Tr_meulage_motif_1_262 := [[-313.7935,-34.766671875,-16.258306640625],[0.588012732058927,-0.500859688362471,0.411836559206125,-0.483498963816164],[0,0,0,0],[8.999999E+09,8.999999E+09,8.999999E+09,8.999999E+09,8.999999E+09,8.999999E+09]];
    LOCAL CONST Robtarget Tr_meulage_motif_1_263 := [[-314.01821875,-33.79225,-16.2588388671875],[0.588012732058927,-0.500859688362471,0.411836559206125,-0.483498963816164],[0,0,0,0],[8.999999E+09,8.999999E+09,8.999999E+09,8.999999E+09,8.999999E+09,8.999999E+09]];
    LOCAL CONST Robtarget Tr_meulage_motif_1_264 := [[-314.2429375,-32.817828125,-16.25937109375],[0.588012732058927,-0.500859688362471,0.411836559206125,-0.483498963816164],[0,0,0,0],[8.999999E+09,8.999999E+09,8.999999E+09,8.999999E+09,8.999999E+09,8.999999E+09]];
    LOCAL CONST Robtarget Tr_meulage_motif_1_265 := [[-314.46765625,-31.843404296875,-16.2599033203125],[0.588012732058927,-0.500859688362471,0.411836559206125,-0.483498963816164],[0,0,0,0],[8.999999E+09,8.999999E+09,8.999999E+09,8.999999E+09,8.999999E+09,8.999999E+09]];
    LOCAL CONST Robtarget Tr_meulage_motif_1_266 := [[-314.692375,-30.868982421875,-16.260435546875],[0.588012732058927,-0.500859688362471,0.411836559206125,-0.483498963816164],[0,0,0,0],[8.999999E+09,8.999999E+09,8.999999E+09,8.999999E+09,8.999999E+09,8.999999E+09]];
    LOCAL CONST Robtarget Tr_meulage_motif_1_267 := [[-314.917125,-29.894560546875,-16.2609677734375],[0.588012732058927,-0.500859688362471,0.411836559206125,-0.483498963816164],[0,0,0,0],[8.999999E+09,8.999999E+09,8.999999E+09,8.999999E+09,8.999999E+09,8.999999E+09]];
    LOCAL CONST Robtarget Tr_meulage_motif_1_268 := [[-315.14184375,-28.920138671875,-16.2615],[0.588012732058927,-0.500859688362471,0.411836559206125,-0.483498963816164],[0,0,0,0],[8.999999E+09,8.999999E+09,8.999999E+09,8.999999E+09,8.999999E+09,8.999999E+09]];
    LOCAL CONST Robtarget Tr_meulage_motif_1_269 := [[-315.3665625,-27.945716796875,-16.2620322265625],[0.588012732058927,-0.500859688362471,0.411836559206125,-0.483498963816164],[0,0,0,0],[8.999999E+09,8.999999E+09,8.999999E+09,8.999999E+09,8.999999E+09,8.999999E+09]];
    LOCAL CONST Robtarget Tr_meulage_motif_1_270 := [[-315.59128125,-26.97129296875,-16.262564453125],[0.588012732058927,-0.500859688362471,0.411836559206125,-0.483498963816164],[0,0,0,0],[8.999999E+09,8.999999E+09,8.999999E+09,8.999999E+09,8.999999E+09,8.999999E+09]];
    LOCAL CONST Robtarget Tr_meulage_motif_1_271 := [[-315.816,-25.99687109375,-16.2630966796875],[0.588012732058927,-0.500859688362471,0.411836559206125,-0.483498963816164],[0,0,0,0],[8.999999E+09,8.999999E+09,8.999999E+09,8.999999E+09,8.999999E+09,8.999999E+09]];
    LOCAL CONST Robtarget Tr_meulage_motif_1_272 := [[-316.04075,-25.02244921875,-16.26362890625],[0.588012732058927,-0.500859688362471,0.411836559206125,-0.483498963816164],[0,0,0,0],[8.999999E+09,8.999999E+09,8.999999E+09,8.999999E+09,8.999999E+09,8.999999E+09]];
    LOCAL CONST Robtarget Tr_meulage_motif_1_273 := [[-316.26546875,-24.04802734375,-16.2641611328125],[0.588012732058927,-0.500859688362471,0.411836559206125,-0.483498963816164],[0,0,0,0],[8.999999E+09,8.999999E+09,8.999999E+09,8.999999E+09,8.999999E+09,8.999999E+09]];
    LOCAL CONST Robtarget Tr_meulage_motif_1_274 := [[-316.4901875,-23.07360546875,-16.2646923828125],[0.588012732058927,-0.500859688362471,0.411836559206125,-0.483498963816164],[0,0,0,0],[8.999999E+09,8.999999E+09,8.999999E+09,8.999999E+09,8.999999E+09,8.999999E+09]];
    LOCAL CONST Robtarget Tr_meulage_motif_1_275 := [[-316.71490625,-22.09918359375,-16.265224609375],[0.588012732058927,-0.500859688362471,0.411836559206125,-0.483498963816164],[0,0,0,0],[8.999999E+09,8.999999E+09,8.999999E+09,8.999999E+09,8.999999E+09,8.999999E+09]];
    LOCAL CONST Robtarget Tr_meulage_motif_1_276 := [[-316.939625,-21.12476171875,-16.2657568359375],[0.588012732058927,-0.500859688362471,0.411836559206125,-0.483498963816164],[0,0,0,0],[8.999999E+09,8.999999E+09,8.999999E+09,8.999999E+09,8.999999E+09,8.999999E+09]];
    LOCAL CONST Robtarget Tr_meulage_motif_1_277 := [[-317.164375,-20.15033984375,-16.2662890625],[0.588012732058927,-0.500859688362471,0.411836559206125,-0.483498963816164],[0,0,0,0],[8.999999E+09,8.999999E+09,8.999999E+09,8.999999E+09,8.999999E+09,8.999999E+09]];
    LOCAL CONST Robtarget Tr_meulage_motif_1_278 := [[-317.38909375,-19.17591796875,-16.2668212890625],[0.588012732058927,-0.500859688362471,0.411836559206125,-0.483498963816164],[0,0,0,0],[8.999999E+09,8.999999E+09,8.999999E+09,8.999999E+09,8.999999E+09,8.999999E+09]];
    LOCAL CONST Robtarget Tr_meulage_motif_1_279 := [[-317.6138125,-18.20149609375,-16.267353515625],[0.588012732058927,-0.500859688362471,0.411836559206125,-0.483498963816164],[0,0,0,0],[8.999999E+09,8.999999E+09,8.999999E+09,8.999999E+09,8.999999E+09,8.999999E+09]];
    LOCAL CONST Robtarget Tr_meulage_motif_1_280 := [[-317.83853125,-17.227072265625,-16.2678857421875],[0.588012732058927,-0.500859688362471,0.411836559206125,-0.483498963816164],[0,0,0,0],[8.999999E+09,8.999999E+09,8.999999E+09,8.999999E+09,8.999999E+09,8.999999E+09]];
    LOCAL CONST Robtarget Tr_meulage_motif_1_281 := [[-318.06325,-16.2526513671875,-16.26841796875],[0.588012732058927,-0.500859688362471,0.411836559206125,-0.483498963816164],[0,0,0,0],[8.999999E+09,8.999999E+09,8.999999E+09,8.999999E+09,8.999999E+09,8.999999E+09]];
    LOCAL CONST Robtarget Tr_meulage_motif_1_282 := [[-318.288,-15.2782294921875,-16.2689501953125],[0.588012732058927,-0.500859688362471,0.411836559206125,-0.483498963816164],[0,0,0,0],[8.999999E+09,8.999999E+09,8.999999E+09,8.999999E+09,8.999999E+09,8.999999E+09]];
    LOCAL CONST Robtarget Tr_meulage_motif_1_283 := [[-318.51271875,-14.303806640625,-16.269482421875],[0.588012732058927,-0.500859688362471,0.411836559206125,-0.483498963816164],[0,0,0,0],[8.999999E+09,8.999999E+09,8.999999E+09,8.999999E+09,8.999999E+09,8.999999E+09]];
    LOCAL CONST Robtarget Tr_meulage_motif_1_284 := [[-318.7374375,-13.329384765625,-16.2700146484375],[0.588012732058927,-0.500859688362471,0.411836559206125,-0.483498963816164],[0,0,0,0],[8.999999E+09,8.999999E+09,8.999999E+09,8.999999E+09,8.999999E+09,8.999999E+09]];
    LOCAL CONST Robtarget Tr_meulage_motif_1_285 := [[-318.96215625,-12.354962890625,-16.270546875],[0.588012732058927,-0.500859688362471,0.411836559206125,-0.483498963816164],[0,0,0,0],[8.999999E+09,8.999999E+09,8.999999E+09,8.999999E+09,8.999999E+09,8.999999E+09]];
    LOCAL CONST Robtarget Tr_meulage_motif_1_286 := [[-319.186875,-11.380541015625,-16.271078125],[0.588012732058927,-0.500859688362471,0.411836559206125,-0.483498963816164],[0,0,0,0],[8.999999E+09,8.999999E+09,8.999999E+09,8.999999E+09,8.999999E+09,8.999999E+09]];
    LOCAL CONST Robtarget Tr_meulage_motif_1_287 := [[-319.411625,-10.406119140625,-16.2716103515625],[0.588012732058927,-0.500859688362471,0.411836559206125,-0.483498963816164],[0,0,0,0],[8.999999E+09,8.999999E+09,8.999999E+09,8.999999E+09,8.999999E+09,8.999999E+09]];
    LOCAL CONST Robtarget Tr_meulage_motif_1_288 := [[-319.63634375,-9.4316962890625,-16.272142578125],[0.588012732058927,-0.500859688362471,0.411836559206125,-0.483498963816164],[0,0,0,0],[8.999999E+09,8.999999E+09,8.999999E+09,8.999999E+09,8.999999E+09,8.999999E+09]];
    LOCAL CONST Robtarget Tr_meulage_motif_1_289 := [[-319.8610625,-8.4572744140625,-16.2726748046875],[0.588012732058927,-0.500859688362471,0.411836559206125,-0.483498963816164],[0,0,0,0],[8.999999E+09,8.999999E+09,8.999999E+09,8.999999E+09,8.999999E+09,8.999999E+09]];
    LOCAL CONST Robtarget Tr_meulage_motif_1_290 := [[-320.08578125,-7.4828525390625,-16.27320703125],[0.588012732058927,-0.500859688362471,0.411836559206125,-0.483498963816164],[0,0,0,0],[8.999999E+09,8.999999E+09,8.999999E+09,8.999999E+09,8.999999E+09,8.999999E+09]];
    LOCAL CONST Robtarget Tr_meulage_motif_1_291 := [[-320.3105,-6.5084306640625,-16.2737392578125],[0.588012732058927,-0.500859688362471,0.411836559206125,-0.483498963816164],[0,0,0,0],[8.999999E+09,8.999999E+09,8.999999E+09,8.999999E+09,8.999999E+09,8.999999E+09]];
    LOCAL CONST Robtarget Tr_meulage_motif_1_292 := [[-320.53525,-5.53400830078125,-16.274271484375],[0.588012732058927,-0.500859688362471,0.411836559206125,-0.483498963816164],[0,0,0,0],[8.999999E+09,8.999999E+09,8.999999E+09,8.999999E+09,8.999999E+09,8.999999E+09]];
    LOCAL CONST Robtarget Tr_meulage_motif_1_293 := [[-320.75996875,-4.55958642578125,-16.2748037109375],[0.588012732058927,-0.500859688362471,0.411836559206125,-0.483498963816164],[0,0,0,0],[8.999999E+09,8.999999E+09,8.999999E+09,8.999999E+09,8.999999E+09,8.999999E+09]];
    LOCAL CONST Robtarget Tr_meulage_motif_1_294 := [[-320.9846875,-3.58516430664063,-16.2753359375],[0.588012732058927,-0.500859688362471,0.411836559206125,-0.483498963816164],[0,0,0,0],[8.999999E+09,8.999999E+09,8.999999E+09,8.999999E+09,8.999999E+09,8.999999E+09]];

